METHOD PROTECTED OnExecErrorClear : DINT
VAR_IN_OUT
  /// Robot assignment of function
  AxesGroup : AxesGroup; 
END_VAR
                  OnExecErrorClear := Reset();
                
END_METHOD

METHOD PROTECTED OnExecRun : DINT
VAR_IN_OUT
  /// Robot assignment of function
  AxesGroup : AxesGroup; 
END_VAR
                  
                
END_METHOD

METHOD PROTECTED OnExecStart : DINT
VAR_IN_OUT
  /// Robot assignment of function
  AxesGroup : AxesGroup; 
END_VAR
                  
                
END_METHOD

METHOD PROTECTED OnUpdateStateFlags
VAR_INPUT
  /// Command message state
  State : CmdMessageState;
END_VAR
                  // Reset State flags
Done := FALSE;

CASE State OF

  // No operation or process is active
  CmdMessageState.EMPTY               :;
  // Created but not yet started
  CmdMessageState.CREATED             :;
  // Buffered and awaiting execution
  CmdMessageState.BUFFERED            :;
  // Buffered in planner for future execution
  CmdMessageState.BUFFERED_IN_PLANNER :;
  // Currently active and in progress
  CmdMessageState.ACTIVE              :;
  // Interrupted and awaiting continuation
  CmdMessageState.INTERRUPTED         :;
  // Requested for abort
  CmdMessageState.ABORT_REQUEST       :;
  // Successfully completed
  CmdMessageState.DONE                : Done := TRUE;
                                        Busy := FALSE;
  // Aborted before completion
  CmdMessageState.ABORTED             : Busy := FALSE;
  // Encountered an error during execution
  CmdMessageState.ERROR               : Error := TRUE;
                                        Busy  := FALSE;
END_CASE
                
END_METHOD

METHOD PROTECTED Reset : DINT
VAR_INPUT
END_VAR
                  Reset := SUPER^.Reset();

Done := FALSE;
Busy := FALSE;
                
END_METHOD
END_FUNCTION_BLOCK

FUNCTION_BLOCK RobotLibraryBaseFB EXTENDS RobotLibraryLogFB
// ------------------------------------------------------------------------- 
//  SRCI Robot Library                                                
// ------------------------------------------------------------------------- 
//                                                                           
//  Object:      RobotLibraryBaseFB                                       
//  Author:      Thorsten Brach                                                
//  Date:        2024-06-01
//
//  Description:                                              
//   
//                                                                           
//  Copyright: 
//    (C) 2024 Thorsten Brach. All rights reserved                                                                                                                                            
//             Licensed under the MIT License.
//                                                                           
//  Disclaimer:                                                                           
//    This project is provided without any guarantee and can be used for   
//    private and commercial purposes. Any use is at the user’s 
//    own risk and responsibility.
//
// -------------------------------------------------------------------------
VAR_INPUT
  /// User defined command name
  Name         : STRING(80);
  /// Execution Mode
  ExecMode     : ExecutionMode;
  /// Priority
  Priority     : PriorityLevel;
END_VAR
VAR_OUTPUT
  /// Command data
  CommandData  : RobotLibraryCommandDataFB;
  /// response data
  ResponseData : RobotLibraryResponseDataFB;
  /// An error occurred during the execution of the command
  Error        : BOOL;
  /// ErrorID reported by RC for error identification according to Table 7-1
  ErrorID      : WORD;
  ErrorIdEnum  : RobotLibraryErrorIdEnum;  
  ErrorAddTxt  : STRING(RobotLibraryConstants.MAX_ADD_TEXT_LENGTH);
  
  /// WarningID for warning identification reported during execution of command according to Table 7-3
  WarningID    : WORD;
  WarningIdEnum: RobotLibraryWarningIdEnum;  
  /// InfoID for info identification reported during execution of command according to Table 7-5
  InfoID       : WORD;    
  InfoIdEnum   : RobotLibraryInfoIdEnum;  
END_VAR
VAR_IN_OUT
  /// Robot assignment of function
  AxesGroup    : AxesGroup; 
END_VAR

VAR
  /// Rising edge for error
  {attribute 'hide'}
 _error_R                  : R_TRIG;
  /// Rising edge for warning
  {attribute 'hide'}
 _warning_R                : R_TRIG;
  /// Rising edge for information
  {attribute 'hide'}
 _info_R                   : R_TRIG;
  /// clear error active
 _clearError               : BOOL;
  /// cancel active
 _cancel                   : BOOL; 
  /// unique ID
 _uniqueID                 : UDINT;  
  /// flag for response received
 _responseReceived         : BOOL;
  /// internal step counter
 _stepCmd                  : DINT;
  /// internal timer  
  {attribute 'hide'}
 _timerCmd                 : TON;
  /// internal timeout 
  {attribute 'hide'}
 _timeoutCmd               : TIME := T#5S;
  /// internal step counter for ClearError
 _stepClearError           : DINT;
  /// internal timer for ClearError
  {attribute 'hide'}
 _timerClearError          : TON;
  /// internal timeout for ClearError 
  {attribute 'hide'}
 _timeoutClearError        : TIME := T#5S;

  /// internal step counter for Cancel
 _stepCancel               : DINT;
  /// internal timer for Cancel  
  {attribute 'hide'}
 _timerCancel              : TON;
  /// internal timeout for Cancel 
  {attribute 'hide'}
 _timeoutCancel            : TIME := T#5S;

  /// internal command header
 _cmdHeader                : CmdHeader;  
  /// internal response header
 _rspHeader                : RspHeader;
  /// internal flag for send a parameter update
 _parameterUpdateInternal  : BOOL; 
  /// internal flag for parameter has changed
 _parameterChanged         : BOOL;
  /// internal flag for parameter are valid
 _parameterValid           : BOOL;
END_VAR

            OnCall               (AxesGroup := AxesGroup);
OnExecRun            (AxesGroup := AxesGroup);
CheckParameterChanged(AxesGroup := AxesGroup);


IF ( AxesGroup.State.OnlineChange_R.Q )
THEN
  OnOnlineChange(AxesGroup := AxesGroup);
END_IF
          

METHOD PUBLIC CallBack : DINT
VAR_INPUT
  /// Response data
  RspData   : AxesGroupAcyclicAcrEntryRspBuffer;  
  /// Timestamp
  Timestamp : SystemTime;
END_VAR
                  // Create log entry
CreateLogMessagePara2 ( Timestamp   := Timestamp,
                        MessageType := MessageType.CMD,
                        Severity    := Severity.DEBUG,
                        MessageCode := 0,
                        MessageText := 'Callback reveiced in FB {1} <{2}>',
                        Para1       := MyType,
                        Para2       := Name);

                   
                   
ResponseData.Reset();
ResponseData.Payload    := RspData.Payload; 
ResponseData.PayloadLen := RspData.PayloadLen;
ParseResponsePayload( ResponseData :=  ResponseData , Timestamp := Timestamp);

// set flag for response received
_responseReceived := TRUE;
                
END_METHOD

METHOD PROTECTED CheckFunctionSupported : BOOL
VAR_IN_OUT
  /// Robot assignment of function
  AxesGroup : AxesGroup; 
END_VAR
                  Error       := TRUE;
ErrorID     := RobotLibraryErrorIdEnum.ERR_FUNCTION_NOT_SUPPORTED;
ErrorAddTxt := CONCAT(THIS^._myType, ' ');
ErrorAddTxt := CONCAT(ErrorAddTxt , THIS^.Name);


// Create log entry
CreateLogMessagePara1 ( Timestamp   := AxesGroup.State.SystemTime,
                        MessageType := MessageType.CMD,
                        Severity    := Severity.DEBUG,
                        MessageCode := 0,
                        MessageText := 'Execution canceled, because function <{1}> is not supported by the robot controller',
                        Para1       :=  _myType);
                
END_METHOD

METHOD PROTECTED CheckParameterChanged : BOOL
VAR_IN_OUT
  /// Robot assignment of function
  AxesGroup    : AxesGroup; 
END_VAR
                  IF ( CheckParameterChanged )
THEN
  AxesGroup.Acyclic.ActiveCommandRegister.NotifyParameterChanged := _uniqueID;
END_IF
                
END_METHOD

METHOD PROTECTED CheckParameterValid : BOOL
VAR_IN_OUT
  /// Robot assignment of function
  AxesGroup : AxesGroup; 
END_VAR
                  CheckParameterValid := TRUE;
                
END_METHOD

METHOD INTERNAL CreateCommandPayload : RobotLibraryCommandDataFB
VAR_IN_OUT
  /// Robot assignment of function
  AxesGroup    : AxesGroup; 
END_VAR
                  // Reset all variables
CreateCommandPayload.Reset();
// Add CmdType
CreateCommandPayload.AddUint(_cmdHeader.CmdTyp);
// Add Reserve_ExecMode
CreateCommandPayload.AddHalfBytes(  0               , _cmdHeader.ExecMode);
// Add ParSeq_Priority
CreateCommandPayload.AddHalfBytes( _cmdHeader.ParSeq, _cmdHeader.Priority);
                
END_METHOD

METHOD PROTECTED OnApplyOutCmd
VAR_INPUT
  /// Command message state
  State : CmdMessageState;
END_VAR
                  
                
END_METHOD

METHOD PROTECTED OnCall
VAR_IN_OUT
  /// Robot assignment of function
  AxesGroup : AxesGroup; 
END_VAR
                  // map numeric value to enum, so that the corresponding message text is directly shown by the tooltip
ErrorIdEnum   := ErrorId;
WarningIdEnum := WarningId;
InfoIdEnum    := InfoId;

Error := ErrorID <> RobotLibraryConstants.OK;

InternalLogger   := AxesGroup.MessageLog; 
ExternalLogger   := AxesGroup.MessageLog.ExternalLogger;
LogLevel         := AxesGroup.MessageLog.LogLevel;

// building rising edges for error, warning, info number detected
_error_R  ( CLK := ErrorID   <> RobotLibraryConstants.OK );
_warning_R( CLK := WarningID <> RobotLibraryConstants.OK );
_info_R   ( CLK := InfoID    <> RobotLibraryConstants.OK );


// Log Command events to message log 
IF  ( LogLevel < _rspHeader.AlarmMessageSeverity ) AND
   (( _error_R  .Q                               ) OR 
    ( _warning_R.Q                               ) OR 
    ( _info_R   .Q                               ))
THEN
  // Add command message to message buffer       
  AxesGroup.MessageLog
    .AddMessageLogByParameter(  Timestamp   :=   AxesGroup.State.SystemTime,
                                MessageType :=   MessageType.CMD,
                                MessageCode :=  _rspHeader.AlarmMessageCode,
                                MessageText :=   CONCAT(MyType, CONCAT(' : ' , MESSAGE_CODE_TO_STRING(_rspHeader.AlarmMessageCode))),
                                Severity    :=  _rspHeader.AlarmMessageSeverity ); 
END_IF 


IF ( _error_R.Q)
THEN
  // Create log entry
  CreateLogMessagePara2 ( Timestamp   := AxesGroup.State.SystemTime,
                          MessageType := MessageType.CMD,
                          Severity    := Severity.DEBUG,
                          MessageCode := 0,
                          MessageText := 'Error with ID: 16#{1} in FB {2} received ',
                          Para1       := WORD_TO_STRING_HEX(ErrorID),
                          Para2       := MyType);                        
END_IF

IF ( _warning_R.Q)
THEN
  // Create log entry
  CreateLogMessagePara2 ( Timestamp   := AxesGroup.State.SystemTime,
                          MessageType := MessageType.CMD,
                          Severity    := Severity.DEBUG,
                          MessageCode := 0,
                          MessageText := 'Warning with ID: 16#{1} in FB {2} received ',
                          Para1       := WORD_TO_STRING_HEX(WarningID),
                          Para2       := MyType);                        
END_IF

IF ( _info_R.Q)
THEN
  // Create log entry
  CreateLogMessagePara2 ( Timestamp   := AxesGroup.State.SystemTime,
                          MessageType := MessageType.CMD,
                          Severity    := Severity.DEBUG,
                          MessageCode := 0,
                          MessageText := 'Info with ID: 16#{1} in FB {2} received ',
                          Para1       := WORD_TO_STRING_HEX(InfoID),
                          Para2       := MyType);                        
END_IF
                
END_METHOD

METHOD PROTECTED OnExecRun : DINT
VAR_IN_OUT
  /// Robot assignment of function
  AxesGroup : AxesGroup; 
END_VAR
                  
                
END_METHOD

METHOD OnOnlineChange : DINT
VAR_IN_OUT
  /// Robot assignment of function
  AxesGroup : AxesGroup; 
END_VAR
                  // update pointer to command FB
AxesGroup.Acyclic.ActiveCommandRegister.OnOnlineChange( UniqueID := _uniqueID, pCommandFB := ADR(THIS^));
                
END_METHOD

METHOD PROTECTED OnUpdateStateFlags
VAR_INPUT
  /// Command message state
  State : CmdMessageState;
END_VAR
                  
                
END_METHOD

METHOD INTERNAL ParseResponsePayload : DINT
VAR_INPUT
  /// Response data
  ResponseData : RobotLibraryResponseDataFB;
  /// Timestamp
  Timestamp    : SystemTime;  
END_VAR
                  // reset message IDs 
InfoID    := 0;
WarningID := 0;
ErrorID   := 0;

// get State
_rspHeader.State                := ResponseData.GetHalfeByte1(IncPayloadPtr := FALSE);
// get ParSeq
_rspHeader.ParSeq               := ResponseData.GetHalfeByte2(IncPayloadPtr := TRUE);
// get AlarmMessageSeverity
_rspHeader.AlarmMessageSeverity := ResponseData.GetSint();
// get AlarmMessageCode
_rspHeader.AlarmMessageCode     := ResponseData.GetUint();


// Update InfoID / WarningID / ErrorID
CASE _rspHeader.AlarmMessageSeverity OF

  // Informative message
  Severity.INFO        : SetInfo   ( InfoID    := _rspHeader.AlarmMessageCode, Overwrite := TRUE );
  // Warning message
  Severity.WARNING     : SetWarning( WarningID := _rspHeader.AlarmMessageCode, Overwrite := TRUE );
  // Error message
  Severity.ERROR       : SetError  ( ErrorID   := _rspHeader.AlarmMessageCode, Overwrite := TRUE ); 
  // Fataö error message
  Severity.FATAL_ERROR : SetError  ( ErrorID   := _rspHeader.AlarmMessageCode, Overwrite := TRUE );

END_CASE

ParseResponsePayload := ResponseData.PayloadPtr;
                
END_METHOD

METHOD PROTECTED Reset : DINT
VAR_INPUT
END_VAR
                  _parameterUpdateInternal := FALSE;
_responseReceived := FALSE;

_uniqueId := 0;
_stepCmd  := 0;
Error     := FALSE;
ErrorID   := 0;
WarningID := 0;
InfoID    := 0;  

Reset := RobotLibraryConstants.OK;
                
END_METHOD

METHOD PUBLIC SetError
VAR_INPUT
  /// ErrorID reported by RC for error identification according to Table 7-1
  ErrorID   : WORD;
  /// TRUE = overwrite an existing error 
  Overwrite : BOOL;
END_VAR
                  IF ( NOT HasError ) OR ( Overwrite )
THEN
  THIS^.ErrorID := ErrorID;
END_IF
                
END_METHOD

METHOD PUBLIC SetInfo
VAR_INPUT
  /// InfoID for info identification reported during execution of command according to Table 7-5
  InfoID    : WORD;
  /// TRUE = overwrite an existing info 
  Overwrite : BOOL;
END_VAR
                  IF ( NOT HasInfo ) OR ( Overwrite )
THEN
  THIS^.InfoID := InfoID;
END_IF
                
END_METHOD

METHOD PUBLIC SetWarning
VAR_INPUT
  /// WarningID for warning identification reported during execution of command according to Table 7-3
  WarningID : WORD;
  /// TRUE = overwrite an existing warning 
  Overwrite : BOOL;
END_VAR
                  IF ( NOT HasWarning ) OR ( Overwrite )
THEN
  THIS^.WarningID := WarningID;
END_IF
                
END_METHOD

PROPERTY PUBLIC HasError : Bool
GET
VAR
END_VAR
                    HasError := ErrorID <> RobotLibraryErrorIdEnum.NO_ERROR;
                  
END_GET
END_PROPERTY

PROPERTY PUBLIC HasInfo : BOOL
GET
VAR
END_VAR
                    HasInfo := InfoID <> RobotLibraryInfoIdEnum.NO_INFO;
                  
END_GET
END_PROPERTY

PROPERTY PUBLIC HasWarning : BOOL
GET
VAR
END_VAR
                    HasWarning := WarningID <> RobotLibraryWarningIdEnum.NO_WARNING;
                  
END_GET
END_PROPERTY
END_FUNCTION_BLOCK

FUNCTION_BLOCK RobotLibraryLogFB
// ------------------------------------------------------------------------- 
//  SRCI Robot Library                                                
// ------------------------------------------------------------------------- 
//                                                                           
//  Object:      RobotLibraryLogFB                                       
//  Author:      Thorsten Brach                                                
//  Date:        2024-11-10
//
//  Description:                                              
//   
//                                                                           
//  Copyright: 
//    (C) 2024 Thorsten Brach. All rights reserved                                                                                                                                            
//             Licensed under the MIT License.
//                                                                           
//  Disclaimer:                                                                           
//    This project is provided without any guarantee and can be used for   
//    private and commercial purposes. Any use is at the user’s 
//    own risk and responsibility.
//
// -------------------------------------------------------------------------
VAR_INPUT
  /// Interface to an internal logger
  InternalLogger : IMessageLogger;  
  /// Interface to an external logger
  ExternalLogger : IMessageLogger;  
  /// Logging level
  LogLevel       : LogLevelEnum := LogLevelEnum.INFO; 
END_VAR

VAR
  /// Type of the function block
 _myType         : STRING;
END_VAR

            
          

METHOD CreateLogMessage : STRING(RobotLibraryParameter.MESSAGE_TEXT_LEN)
VAR_INPUT
  /// Timestamp
  Timestamp   : SystemTime;
  /// Type of message according to Table 5-46:
  MessageType : MessageType;
  /// Severity of message according to Table 5-47: Debug, Info, Warning, Error, Fatal error
  Severity    : Severity;
  /// Code of messages
  MessageCode : DWORD;
  /// Static text of message
  MessageText : STRING(RobotLibraryParameter.MESSAGE_TEXT_LEN);  
END_VAR

VAR
  /// internal log message 
 _message    : AlarmMessage;
  /// internal string
 _tmpString  : STRING(255);
END_VAR
                  IF ( LogLevel <= Severity )
THEN
 _message.Timestamp   := Timestamp;
 _message.MessageType := MessageType;
 _message.Severity    := Severity;
 _message.MessageCode := MessageCode;
 _message.MessageText := StrPadRight(MyType,' ', RobotLibraryDefines.MaxTypeNameLength);
 _message.MessageText := CONCAT(_message.MessageText, ': ');
 _message.MessageText := CONCAT(_message.MessageText,MessageText);

  // return log message
  CreateLogMessage := ALARM_MESSAGE_TO_STRING(_message);
  
  // Check internal logger valid ? 
  IF ( InternalLogger <> 0 )
  THEN  
    InternalLogger.AddSystemLog( SystemLog := ALARM_MESSAGE_TO_STRING(_message));
  END_IF

  // Check external logger valid ? 
  IF ( ExternalLogger <> 0 )
  THEN  
    ExternalLogger.AddSystemLog( SystemLog := ALARM_MESSAGE_TO_STRING(_message));
  END_IF
END_IF
                
END_METHOD

METHOD CreateLogMessagePara1 : STRING(RobotLibraryParameter.MESSAGE_TEXT_LEN)
VAR_INPUT
  /// Timestamp
  Timestamp   : SystemTime;
  /// Type of message according to Table 5-46:
  MessageType : MessageType;
  /// Severity of message according to Table 5-47: Debug, Info, Warning, Error, Fatal error
  Severity    : Severity;
  /// Code of messages
  MessageCode : DWORD;
  /// Static text of message
  MessageText : STRING(RobotLibraryParameter.MESSAGE_TEXT_LEN);  
  /// sub string which will replace the placeholder {1}
  Para1       : STRING(RobotLibraryParameter.MESSAGE_TEXT_LEN);
END_VAR
VAR
  /// internal log message 
 _logMessage : AlarmMessage;
END_VAR
                  IF ( LogLevel <= Severity )
THEN
  MessageText := StrReplace(MessageText,'{1}', Para1);
  
  CreateLogMessagePara1 
    := CreateLogMessage( Timestamp   := Timestamp,
                         MessageType := MessageType,
                         Severity    := Severity,
                         MessageCode := MessageCode,
                         MessageText := MessageText);
END_IF                         
                
END_METHOD

METHOD CreateLogMessagePara2 : STRING(RobotLibraryParameter.MESSAGE_TEXT_LEN)
VAR_INPUT
  /// Timestamp
  Timestamp   : SystemTime;
  /// Type of message according to Table 5-46:
  MessageType : MessageType;
  /// Severity of message according to Table 5-47: Debug, Info, Warning, Error, Fatal error
  Severity    : Severity;
  /// Code of messages
  MessageCode : DWORD;
  /// Static text of message
  MessageText : STRING(RobotLibraryParameter.MESSAGE_TEXT_LEN);  
  /// sub string which will replace the placeholder {1}
  Para1       : STRING(RobotLibraryParameter.MESSAGE_TEXT_LEN);
  /// sub string which will replace the placeholder {2}
  Para2       : STRING(RobotLibraryParameter.MESSAGE_TEXT_LEN);
END_VAR
VAR
  /// internal log message 
 _logMessage : AlarmMessage;
END_VAR
                  IF ( LogLevel <= Severity )
THEN
  MessageText := StrReplace(MessageText,'{2}', Para2);
  
  CreateLogMessagePara2 
    := CreateLogMessagePara1( Timestamp   := Timestamp,
                              MessageType := MessageType,
                              Severity    := Severity,
                              MessageCode := MessageCode,
                              MessageText := MessageText,
                              Para1       := Para1);
END_IF                              
                
END_METHOD

METHOD CreateLogMessagePara3 : STRING(RobotLibraryParameter.MESSAGE_TEXT_LEN)
VAR_INPUT
  /// Timestamp
  Timestamp   : SystemTime;
  /// Type of message according to Table 5-46:
  MessageType : MessageType;
  /// Severity of message according to Table 5-47: Debug, Info, Warning, Error, Fatal error
  Severity    : Severity;
  /// Code of messages
  MessageCode : DWORD;
  /// Static text of message
  MessageText : STRING(RobotLibraryParameter.MESSAGE_TEXT_LEN);  
  /// sub string which will replace the placeholder {1}
  Para1       : STRING(RobotLibraryParameter.MESSAGE_TEXT_LEN);
  /// sub string which will replace the placeholder {2}
  Para2       : STRING(RobotLibraryParameter.MESSAGE_TEXT_LEN);
  /// sub string which will replace the placeholder {3}
  Para3       : STRING(RobotLibraryParameter.MESSAGE_TEXT_LEN);
END_VAR
VAR
  /// internal log message 
 _logMessage : AlarmMessage;
END_VAR
                  IF ( LogLevel <= Severity )
THEN
  MessageText := StrReplace(MessageText,'{3}', Para3);
  
  CreateLogMessagePara3
    := CreateLogMessagePara2( Timestamp   := Timestamp,
                              MessageType := MessageType,
                              Severity    := Severity,
                              MessageCode := MessageCode,
                              MessageText := MessageText,
                              Para1       := Para1,
                              Para2       := Para2);
END_IF                              
                
END_METHOD

METHOD CreateLogMessagePara4 : STRING(RobotLibraryParameter.MESSAGE_TEXT_LEN)
VAR_INPUT
  /// Timestamp
  Timestamp   : SystemTime;
  /// Type of message according to Table 5-46:
  MessageType : MessageType;
  /// Severity of message according to Table 5-47: Debug, Info, Warning, Error, Fatal error
  Severity    : Severity;
  /// Code of messages
  MessageCode : DWORD;
  /// Static text of message
  MessageText : STRING(RobotLibraryParameter.MESSAGE_TEXT_LEN);  
  /// sub string which will replace the placeholder {1}
  Para1       : STRING(RobotLibraryParameter.MESSAGE_TEXT_LEN);
  /// sub string which will replace the placeholder {2}
  Para2       : STRING(RobotLibraryParameter.MESSAGE_TEXT_LEN);
  /// sub string which will replace the placeholder {3}
  Para3       : STRING(RobotLibraryParameter.MESSAGE_TEXT_LEN);
  /// sub string which will replace the placeholder {4}
  Para4       : STRING(RobotLibraryParameter.MESSAGE_TEXT_LEN);
END_VAR
VAR
  /// internal log message 
 _logMessage : AlarmMessage;
END_VAR
                  IF ( LogLevel <= Severity )
THEN
  MessageText := StrReplace(MessageText,'{4}', Para4);
  
  CreateLogMessagePara4
    := CreateLogMessagePara3( Timestamp   := Timestamp,
                              MessageType := MessageType,
                              Severity    := Severity,
                              MessageCode := MessageCode,
                              MessageText := MessageText,
                              Para1       := Para1,
                              Para2       := Para2,
                              Para3       := Para3);
END_IF                              
                
END_METHOD

METHOD CreateLogMessagePara5 : STRING(RobotLibraryParameter.MESSAGE_TEXT_LEN)
VAR_INPUT
  /// Timestamp
  Timestamp   : SystemTime;
  /// Type of message according to Table 5-46:
  MessageType : MessageType;
  /// Severity of message according to Table 5-47: Debug, Info, Warning, Error, Fatal error
  Severity    : Severity;
  /// Code of messages
  MessageCode : DWORD;
  /// Static text of message
  MessageText : STRING(RobotLibraryParameter.MESSAGE_TEXT_LEN);  
  /// sub string which will replace the placeholder {1}
  Para1       : STRING(RobotLibraryParameter.MESSAGE_TEXT_LEN);
  /// sub string which will replace the placeholder {2}
  Para2       : STRING(RobotLibraryParameter.MESSAGE_TEXT_LEN);
  /// sub string which will replace the placeholder {3}
  Para3       : STRING(RobotLibraryParameter.MESSAGE_TEXT_LEN);
  /// sub string which will replace the placeholder {4}
  Para4       : STRING(RobotLibraryParameter.MESSAGE_TEXT_LEN);
  /// sub string which will replace the placeholder {5}
  Para5       : STRING(RobotLibraryParameter.MESSAGE_TEXT_LEN);
END_VAR
VAR
  /// internal log message 
 _logMessage : AlarmMessage;
END_VAR
                  IF ( LogLevel <= Severity )
THEN  
  MessageText := StrReplace(MessageText,'{5}', Para5);
  
  CreateLogMessagePara5
    := CreateLogMessagePara4( Timestamp   := Timestamp,
                              MessageType := MessageType,
                              Severity    := Severity,
                              MessageCode := MessageCode,
                              MessageText := MessageText,
                              Para1       := Para1,
                              Para2       := Para2,
                              Para3       := Para3,
                              Para4       := Para4);
END_IF                              
                
END_METHOD

METHOD CreateLogMessagePara6 : STRING(RobotLibraryParameter.MESSAGE_TEXT_LEN)
VAR_INPUT
  /// Timestamp
  Timestamp   : SystemTime;
  /// Type of message according to Table 5-46:
  MessageType : MessageType;
  /// Severity of message according to Table 5-47: Debug, Info, Warning, Error, Fatal error
  Severity    : Severity;
  /// Code of messages
  MessageCode : DWORD;
  /// Static text of message
  MessageText : STRING(RobotLibraryParameter.MESSAGE_TEXT_LEN);  
  /// sub string which will replace the placeholder {1}
  Para1       : STRING(RobotLibraryParameter.MESSAGE_TEXT_LEN);
  /// sub string which will replace the placeholder {2}
  Para2       : STRING(RobotLibraryParameter.MESSAGE_TEXT_LEN);
  /// sub string which will replace the placeholder {3}
  Para3       : STRING(RobotLibraryParameter.MESSAGE_TEXT_LEN);
  /// sub string which will replace the placeholder {4}
  Para4       : STRING(RobotLibraryParameter.MESSAGE_TEXT_LEN);
  /// sub string which will replace the placeholder {5}
  Para5       : STRING(RobotLibraryParameter.MESSAGE_TEXT_LEN);
  /// sub string which will replace the placeholder {6}
  Para6       : STRING(RobotLibraryParameter.MESSAGE_TEXT_LEN);
END_VAR
VAR
  /// internal log message 
 _logMessage : AlarmMessage;
END_VAR
                  IF ( LogLevel <= Severity )
THEN
  MessageText := StrReplace(MessageText,'{6}', Para6);
  
  CreateLogMessagePara6
    := CreateLogMessagePara5( Timestamp   := Timestamp,
                              MessageType := MessageType,
                              Severity    := Severity,
                              MessageCode := MessageCode,
                              MessageText := MessageText,
                              Para1       := Para1,
                              Para2       := Para2,
                              Para3       := Para3,
                              Para4       := Para4,
                              Para5       := Para5);
END_IF                       
                
END_METHOD

PROPERTY PROTECTED MyType : STRING
GET
VAR
END_VAR
                    MyType := _myType;
                  
END_GET
SET
VAR
END_VAR
                    _myType := MyType;

// set the max type name length 
RobotLibraryDefines.MaxTypeNameLength := MAX(LEN(_myType), RobotLibraryDefines.MaxTypeNameLength);
                  
END_SET
END_PROPERTY
END_FUNCTION_BLOCK

FUNCTION_BLOCK AxesGroupMessageLogFB IMPLEMENTS IMessageLogger
// ------------------------------------------------------------------------- 
//  SRCI Robot Library                                                
// ------------------------------------------------------------------------- 
//                                                                           
//  Object:      AxesGroupMessageLogFB                                       
//  Author:      Thorsten Brach                                                
//  Date:        2025-01-05
//
//  Description:                                              
//   
//                                                                           
//  Copyright: 
//    (C) 2025 Thorsten Brach. All rights reserved                                                                                                                                            
//             Licensed under the MIT License.
//                                                                           
//  Disclaimer:                                                                           
//    This project is provided without any guarantee and can be used for   
//    private and commercial purposes. Any use is at the user’s 
//    own risk and responsibility.
//
// -------------------------------------------------------------------------
VAR_INPUT
  /// Logging level
  LogLevel         : LogLevel;
  /// Interface to an external logger
  ExternalLogger   : IMessageLogger;
END_VAR


VAR_OUTPUT
  /// Amount of system log entries
  SystemLogEntries : UINT := 0;
  /// Amount of message log entries
  MessagesEntries  : UINT := 0;
  /// System log
  SystemLogs       : ARRAY[0..RobotLibraryParameter.SYSTEM_LOG_MAX ] OF STRING(RobotLibraryParameter.MESSAGE_TEXT_LEN);
  /// Message Log
  Messages         : ARRAY[0..RobotLibraryParameter.MESSAGE_LOG_MAX] OF AlarmMessage;  
END_VAR

            
          

METHOD PUBLIC AddMessageLog
VAR_INPUT
  MessageLog : AlarmMessage;
END_VAR

VAR
  /// internal index
 _idx            : DINT;
  /// internal index to delete
 _idxFound       : DINT;
  /// lowest Severity
 _lowestSeverity : Severity := Severity.FATAL_ERROR;
  /// temporary buffer ( must be one element less than the message log !!! )
 _tmpBuffer      : ARRAY[0..RobotLibraryParameter.MESSAGE_LOG_MAX -1] OF AlarmMessage; 
END_VAR
                  // Check entry must be added ? 
IF (( LogLevel  <= MessageLog.Severity     ) AND
    ( LogLevel  >  LogLevelEnum.DEACTIVATE ))
THEN
  // Check message buffer is full ? 
  IF ( MessagesEntries >= RobotLibraryParameter.MESSAGE_LOG_MAX )
  THEN
    // find lowest Severity
    FOR _idx := 1 TO RobotLibraryParameter.MESSAGE_LOG_MAX
    DO
      // check entry has a lower severity ? 
     _lowestSeverity := MIN( Messages[_idx].Severity, _lowestSeverity );
		END_FOR

    // search for the oldes message with a lower Severity 
    FOR _idx := RobotLibraryParameter.MESSAGE_LOG_MAX TO 1 BY -1
    DO
      // message found ?
      IF (( Messages[_idx].Severity <   MessageLog.Severity ) AND
          ( Messages[_idx].Severity <= _lowestSeverity      ))
      THEN
        // save index to delete 
       _idxFound := _idx;
        EXIT;
			END_IF
		END_FOR
    
    // check message must be deleted ? 
    IF ( _idxFound > 0 )
    THEN
      // shift all messages starting from the found index one position forwards
      FOR _idx := _idxFound TO RobotLibraryParameter.MESSAGE_LOG_MAX -1
      DO
        Messages[_idx] := Messages[_idx +1];
			END_FOR
		END_IF
  END_IF  

  // shift all messages one position backwards
  // shift messages log entries
  SysDepMemCpy( pDest := ADR(_tmpBuffer[0]), pSrc := ADR(  Messages[0]), DataLen := SIZEOF(_tmpBuffer));
  SysDepMemCpy( pDest := ADR(  Messages[1]), pSrc := ADR(_tmpBuffer[0]), DataLen := SIZEOF(_tmpBuffer));
  
  
  // Add new message 
  Messages[0].Timestamp   := MessageLog.Timestamp;           
  Messages[0].MessageType := MessageLog.MessageType;
  Messages[0].Severity    := MessageLog.Severity;
  Messages[0].MessageText := MessageLog.MessageText;
  Messages[0].MessageCode := MessageLog.MessageCode;
  
  // inc message counter
  MessagesEntries := DINT_TO_UINT(LIMIT(0, MessagesEntries + 1, RobotLibraryParameter.MESSAGE_LOG_MAX));
END_IF
                
END_METHOD

METHOD Public AddMessageLogByParameter
VAR_INPUT
  /// Timestamp
  Timestamp   : SystemTime;
  /// Type of message according to Table 5-46:
  MessageType : MessageType;
  /// Severity of message according to Table 5-47: Debug, Info, Warning, Error, Fatal error
  Severity    : Severity;
  /// Code of messages
  MessageCode : DWORD;
  /// Static text of message
  MessageText : STRING(RobotLibraryParameter.MESSAGE_TEXT_LEN);    
END_VAR

VAR
  /// temporary message 
 _message : AlarmMessage;
END_VAR
                  _message.Timestamp   := Timestamp;
_message.MessageType := MessageType;
_message.MessageCode := MessageCode;
_message.MessageText := MessageText;
_message.Severity    := Severity;

// Add message to message buffer       
AddMessageLog(_message);        
                
END_METHOD

METHOD PUBLIC AddSystemLog
VAR_INPUT
  /// system log message
  SystemLog : STRING(255);
END_VAR
VAR
  /// internal index
 _idx       : DINT;
  /// internal log message 
 _message   : AlarmMessage;
  /// temporary buffer ( must be one element less than the system log !!! )
 _tmpBuffer : ARRAY[0..RobotLibraryParameter.SYSTEM_LOG_MAX -1] OF STRING(RobotLibraryParameter.MESSAGE_TEXT_LEN);
END_VAR
                  // shift system log entries
SysDepMemCpy( pDest := ADR(_tmpBuffer[0]), pSrc := ADR(SystemLogs[0]), DataLen := SIZEOF(_tmpBuffer));
SysDepMemCpy( pDest := ADR(SystemLogs[1]), pSrc := ADR(_tmpBuffer[0]), DataLen := SIZEOF(_tmpBuffer));

// Delete CR from system log message
SystemLog := StrReplace(SystemLog, '$R', '');
// Delete LF from system log message          
SystemLog := StrReplace(SystemLog, '$N', '');    
       
// Add System log to buffer 
SystemLogs[0] := SystemLog;
 
// inc SystemLog counter
SystemLogEntries := DINT_TO_UINT(LIMIT(0, SystemLogEntries + 1, RobotLibraryParameter.SYSTEM_LOG_MAX));
                
END_METHOD

METHOD CheckMessageCodePresent : BOOL
VAR_INPUT
  /// Code of messages
  MessageCode : DWORD;
END_VAR

VAR
  /// internal index for loops
 _idx : DINT;
END_VAR
                  FOR _idx := 0 TO RobotLibraryParameter.MESSAGE_LOG_MAX
DO
  IF (Messages[_idx].MessageCode = MessageCode)
  THEN
    CheckMessageCodePresent := TRUE;
    RETURN;
	END_IF
END_FOR
                
END_METHOD

METHOD PUBLIC DeleteMessages
VAR_INPUT
END_VAR
                  // reset messages
SysDepMemSet(ADR(Messages), 0, SIZEOF(Messages));
// reset message counter
MessagesEntries := 0;
                
END_METHOD

METHOD DeleteSystemLogs
VAR_INPUT
END_VAR
                  // reset SystemLogs
SysDepMemSet(ADR(SystemLogs), 0, SIZEOF(SystemLogs));
// reset SystemLogs counter
SystemLogEntries := 0;
                
END_METHOD
END_FUNCTION_BLOCK

{attribute 'pack_mode' := '1'} 
FUNCTION_BLOCK RobotLibraryRecvDataBaseFB
// ------------------------------------------------------------------------- 
//  SRCI Robot Library                                                
// ------------------------------------------------------------------------- 
//                                                                           
//  Object:      RobotLibraryRecvDataFB                                       
//  Author:      Thorsten Brach                                                
//  Date:        2024-06-01
//
//  Description:                                              
//   
//                                                                           
//  Copyright: 
//    (C) 2024 Thorsten Brach. All rights reserved                                                                                                                                            
//             Licensed under the MIT License.
//                                                                           
//  Disclaimer:                                                                           
//    This project is provided without any guarantee and can be used for   
//    private and commercial purposes. Any use is at the user’s 
//    own risk and responsibility.
//
// -------------------------------------------------------------------------
VAR_INPUT
  /// Payload length
  PayloadLen : UDINT;
  /// Payload pointer
  PayloadPtr : DINT;
END_VAR

VAR
  /// internal pointer to payload 
  pPayload : POINTER TO BYTE;
END_VAR

            
          

/// returns a ArmConfigParameter from the payload buffer from the current payload pointer address and increase the payload pointer afterwards
METHOD GetArmConfig : ArmConfigParameter
VAR
  /// temporary byte
 _tmpByte : BYTE;
END_VAR
// Table 5-17: Meaning of “Config” byte
// BIT 0 Shoulder TRUE : Shoulder is Back
//                FALSE: Shoulder is Front
// BIT 1 Elbow    TRUE : Elbow is Down
//                FALSE: Elbow is Up
// BIT 2 Wrist    TRUE : Wrist is Flip
//                FALSE: Wrist is Non-Flip
// BIT 3 Spare Not used
// BIT 4 Spare Not Used
// BIT 5 Spare Not Used
// BIT 6 Spare Not Used
// BIT 7 Spare Not Used
                  // get 1st Byte
_tmpByte := GetByte();

IF ( _tmpByte.0 ) 
THEN
  GetArmConfig.Shoulder := ArmConfigShoulder.BACK;
ELSE
  GetArmConfig.Shoulder := ArmConfigShoulder.FRONT;
END_IF

IF ( _tmpByte.1 ) 
THEN
  GetArmConfig.Elbow := ArmConfigElbow.DOWN;
ELSE
  GetArmConfig.Elbow := ArmConfigElbow.UP;
END_IF

IF ( _tmpByte.2 ) 
THEN
  GetArmConfig.Wrist := ArmConfigWrist.FLIP;
ELSE
  GetArmConfig.Wrist := ArmConfigWrist.NON_FLIP;
END_IF


// get 2nd byte to inc the PayloadPointer
_tmpByte := GetByte();
                
END_METHOD

/// returns a BOOL from the payload buffer from the current payload pointer address and increase the payload pointer afterwards
METHOD GetBool : BOOL
VAR
  /// temporary byte
  _tmpByte : BYTE;
END_VAR
                  // update internal pointer
UpdatePointer();

// check pointer is valid ? 
IF (pPayload = RobotLibraryConstants.NULL_POINTER)
THEN
  RETURN;
END_IF


_tmpByte := GetByte();

// copy data
GetBool := _tmpByte.0;

                
END_METHOD

/// returns a BYTE from the payload buffer from the current payload pointer address and increase the payload pointer afterwards
METHOD GetByte : BYTE
VAR
  /// internal pointer to byte
  _tmpPointer : POINTER TO BYTE;
END_VAR
                  // update internal pointer
UpdatePointer();

// check pointer is valid ? 
IF (pPayload = RobotLibraryConstants.NULL_POINTER)
THEN
  RETURN;
END_IF


_tmpPointer := pPayload + DINT_TO_DWORD(PayloadPtr);

// copy data
GetByte := _tmpPointer^;
// inc payload pointer 
PayloadPtr := PayloadPtr + SIZEOF(BYTE);
                
END_METHOD

/// returns a datablock from the payload buffer from the current payload pointer address and increase the payload pointer afterwards
METHOD GetDataBlock
VAR_INPUT
  /// Target
  pData    : POINTER TO BYTE;
  /// Size of data block
  Size     : UDINT;
  /// Target data type is string ? 
  IsString : BOOL;
END_VAR
                  // update internal pointer
UpdatePointer();

// check pointer is valid ? 
IF (pPayload = RobotLibraryConstants.NULL_POINTER)
THEN
  RETURN;
END_IF


IF ( pData <> RobotLibraryConstants.NULL_POINTER)
THEN
  IF ( IsString)
  THEN
    Size := Size -1;
  END_IF

  // copy data
  SysDepMemCpy(pDest := pData, pSrc := pPayload + DINT_TO_DWORD(PayloadPtr), DataLen := Size);
  
  // inc payload pointer 
  PayloadPtr := PayloadPtr + UDINT_TO_DINT(Size);
END_IF
                
END_METHOD

/// returns a DataInSync from the payload buffer from the current payload pointer address and increase the payload pointer afterwards
METHOD GetDataInSync : DataInSync
VAR
  /// temporary byte
 _tmpByte : BYTE;
END_VAR
                  // update internal pointer
UpdatePointer();

// check pointer is valid ? 
IF (pPayload = RobotLibraryConstants.NULL_POINTER)
THEN
  RETURN;
END_IF


// copy data
_tmpByte := GetByte();

GetDataInSync.ToolsInSync             := _tmpByte.0;
GetDataInSync.FramesInSync            := _tmpByte.1;
GetDataInSync.LoadsInSync             := _tmpByte.2;
GetDataInSync.WorkAreasInSync         := _tmpByte.3;
GetDataInSync.SoftwareLimitsInSync    := _tmpByte.4;
GetDataInSync.DefaultDynamicsInSync   := _tmpByte.5;
GetDataInSync.ReferenceDynamicsInSync := _tmpByte.6;
                
END_METHOD

/// returns a DWORD from the payload buffer from the current payload pointer address and increase the payload pointer afterwards
METHOD GetDword : DWORD
                  // update internal pointer
UpdatePointer();

// check pointer is valid ? 
IF (pPayload = RobotLibraryConstants.NULL_POINTER)
THEN
  RETURN;
END_IF

// copy data
SysDepMemCpy(pDest := ADR(GetDword), pSrc := pPayload + DINT_TO_DWORD(PayloadPtr), DataLen := SIZEOF(DWORD));
// inc payload pointer 
PayloadPtr := PayloadPtr + SIZEOF(DWORD);
                
END_METHOD

/// returns a FragmentAction from the payload buffer from the current payload pointer address and increase the payload pointer afterwards
METHOD GetFragmentAction : FragmentAction
VAR
  /// temporary byte
 _tmpByte : BYTE;
END_VAR
                  // update internal pointer
UpdatePointer();

// check pointer is valid ? 
IF (pPayload = RobotLibraryConstants.NULL_POINTER)
THEN
  RETURN;
END_IF

// copy data
_tmpByte := GetByte();

GetFragmentAction.Complete := _tmpByte.0;
GetFragmentAction.Reset    := _tmpByte.1;
GetFragmentAction.Clear    := _tmpByte.2;
GetFragmentAction.BIT03    := _tmpByte.3;
GetFragmentAction.BIT04    := _tmpByte.4;
GetFragmentAction.BIT05    := _tmpByte.5;
GetFragmentAction.BIT06    := _tmpByte.6;
GetFragmentAction.BIT07    := _tmpByte.7;

                
END_METHOD

/// returns the 1st halfe BYTE from the payload buffer from the current payload pointer address and increase the payload pointer afterwards
METHOD GetHalfeByte1 : BYTE
VAR_INPUT
  /// Increase payload pointer 
  IncPayloadPtr : BOOL;
END_VAR

VAR
  /// temporary byte
 _tmpByte    : BYTE;
  /// internal pointer to byte
 _tmpPointer : POINTER TO BYTE;
END_VAR
                  // update internal pointer
UpdatePointer();

// check pointer is valid ? 
IF (pPayload = RobotLibraryConstants.NULL_POINTER)
THEN
  RETURN;
END_IF

// set pointer
_tmpPointer := pPayload + DINT_TO_DWORD(PayloadPtr); 
// copy data
_tmpByte := _tmpPointer^;

GetHalfeByte1.0 := _tmpByte.0;
GetHalfeByte1.1 := _tmpByte.1;
GetHalfeByte1.2 := _tmpByte.2;
GetHalfeByte1.3 := _tmpByte.3;

IF (IncPayloadPtr)
THEN  
  // inc payload pointer
  PayloadPtr := PayloadPtr + SIZEOF(BYTE);
END_IF
                
END_METHOD

/// returns the 1st halfe BYTE from the payload buffer from the current payload pointer address and increase the payload pointer afterwards
METHOD GetHalfeByte2 : BYTE
VAR_INPUT
  /// Increase payload pointer 
  IncPayloadPtr : BOOL;
END_VAR

VAR
  /// temporary byte
 _tmpByte    : BYTE;
  /// internal pointer to byte
 _tmpPointer : POINTER TO BYTE;
END_VAR
                  // update internal pointer
UpdatePointer();

// check pointer is valid ? 
IF (pPayload = RobotLibraryConstants.NULL_POINTER)
THEN
  RETURN;
END_IF

// set pointer
_tmpPointer := pPayload + DINT_TO_DWORD(PayloadPtr); 
// copy data
_tmpByte := _tmpPointer^;

GetHalfeByte2.0 := _tmpByte.4;
GetHalfeByte2.1 := _tmpByte.5;
GetHalfeByte2.2 := _tmpByte.6;
GetHalfeByte2.3 := _tmpByte.7;

IF (IncPayloadPtr)
THEN  
  // inc payload pointer
  PayloadPtr := PayloadPtr + SIZEOF(BYTE);
END_IF

                
END_METHOD

/// returns a IEC_Date from the payload buffer from the current payload pointer address and increase the payload pointer afterwards
METHOD GetIecDate : IEC_Date
                  // update internal pointer
UpdatePointer();

// check pointer is valid ? 
IF (pPayload = RobotLibraryConstants.NULL_POINTER)
THEN
  RETURN;
END_IF

// copy data
SysDepMemCpy(pDest := ADR(GetIecDate), pSrc := pPayload + DINT_TO_DWORD(PayloadPtr), DataLen := SIZEOF(IEC_DATE));
// swap byte order
GetIecDate := SwapIecDate(GetIecDate);
// inc payload pointer   
PayloadPtr := PayloadPtr + SIZEOF(IEC_DATE);
                
END_METHOD

/// returns a IEC_TIME from the payload buffer from the current payload pointer address and increase the payload pointer afterwards
METHOD GetIecTime : IEC_TIME
                  // update internal pointer
UpdatePointer();

// check pointer is valid ? 
IF (pPayload = RobotLibraryConstants.NULL_POINTER)
THEN
  RETURN;
END_IF

// copy data
SysDepMemCpy(pDest := ADR(GetIecTime), pSrc := pPayload + DINT_TO_DWORD(PayloadPtr), DataLen := SIZEOF(IEC_TIME));
// swap byte order
GetIecTime := SwapIecTime(GetIecTime);
// inc payload pointer   
PayloadPtr := PayloadPtr + SIZEOF(IEC_TIME);
                
END_METHOD

/// returns a INT from the payload buffer from the current payload pointer address and increase the payload pointer afterwards
METHOD GetInt : INT
                  // update internal pointer
UpdatePointer();

// check pointer is valid ? 
IF (pPayload = RobotLibraryConstants.NULL_POINTER)
THEN
  RETURN;
END_IF

// copy data
SysDepMemCpy(pDest := ADR(GetInt), pSrc := pPayload + DINT_TO_DWORD(PayloadPtr), DataLen := SIZEOF(INT));
// swap byte order
GetInt := SwapInt(GetInt);
// inc payload pointer   
PayloadPtr := PayloadPtr + SIZEOF(INT);
                
END_METHOD

/// returns a REAL from the payload buffer from the current payload pointer address and increase the payload pointer afterwards
METHOD GetReal : REAL
                  // update internal pointer
UpdatePointer();

// check pointer is valid ? 
IF (pPayload = RobotLibraryConstants.NULL_POINTER)
THEN
  RETURN;
END_IF

// copy data
SysDepMemCpy(pDest := ADR(GetReal), pSrc := pPayload + DINT_TO_DWORD(PayloadPtr), DataLen := SIZEOF(REAL));
// swap byte order
GetReal := SwapReal(GetReal);
// inc payload pointer   
PayloadPtr := PayloadPtr + SIZEOF(Real);
                
END_METHOD

/// returns a SINT from the payload buffer from the current payload pointer address and increase the payload pointer afterwards
METHOD GetSint : SINT
                  // update internal pointer
UpdatePointer();

// check pointer is valid ? 
IF (pPayload = RobotLibraryConstants.NULL_POINTER)
THEN
  RETURN;
END_IF

// copy data
SysDepMemCpy(pDest := ADR(GetSint), pSrc := pPayload + DINT_TO_DWORD(PayloadPtr), DataLen := SIZEOF(SINT));
// inc payload pointer 
PayloadPtr := PayloadPtr + SIZEOF(SINT);
                
END_METHOD

/// returns a String from the payload buffer from the current payload pointer address and increase the payload pointer afterwards
METHOD GetString : STRING(255)
VAR_INPUT
  Size : DINT;
END_VAR
                  // update internal pointer
UpdatePointer();

// check pointer is valid ? 
IF (pPayload = RobotLibraryConstants.NULL_POINTER)
THEN
  RETURN;
END_IF

// copy data
SysDepMemCpy(pDest := ADR(GetString), pSrc := pPayload + DINT_TO_DWORD(PayloadPtr), DataLen := DINT_TO_UDINT(Size));

// inc payload pointer 
PayloadPtr := PayloadPtr + Size;
                
END_METHOD

/// returns a TrackingStatus from the payload buffer from the current payload pointer address and increase the payload pointer afterwards
METHOD GetTrackingStatus : TrackingStatus
VAR
  /// temporary byte
  tmpByte : BYTE;
END_VAR
                  // update internal pointer
UpdatePointer();

// check pointer is valid ? 
IF (pPayload = RobotLibraryConstants.NULL_POINTER)
THEN
  RETURN;
END_IF

// copy data
tmpByte := GetByte();

GetTrackingStatus.ConveyorTrackingEnabled   := tmpByte.0;  
GetTrackingStatus.WaitingForSynchronization := tmpByte.1;
GetTrackingStatus.Synchronizing             := tmpByte.2;
GetTrackingStatus.Synchronous               := tmpByte.3;
GetTrackingStatus.Desynchronizing           := tmpByte.4;
GetTrackingStatus.SyncOutZoneEntered        := tmpByte.5;
GetTrackingStatus.SyncOutZoneLeft           := tmpByte.6;
GetTrackingStatus.NotUsed                   := tmpByte.7;   
                
END_METHOD

/// returns a TurnNumber from the payload buffer from the current payload pointer address and increase the payload pointer afterwards
METHOD GetTurnNumbers : TurnNumber
                  // update internal pointer
UpdatePointer();

// check pointer is valid ? 
IF (pPayload = RobotLibraryConstants.NULL_POINTER)
THEN
  RETURN;
END_IF

GetTurnNumbers.J1Turns := BYTE_TO_SINT(GetHalfeByte1(FALSE));
GetTurnNumbers.J2Turns := BYTE_TO_SINT(GetHalfeByte2(TRUE));

GetTurnNumbers.J3Turns := BYTE_TO_SINT(GetHalfeByte1(FALSE));
GetTurnNumbers.J4Turns := BYTE_TO_SINT(GetHalfeByte2(TRUE));

GetTurnNumbers.J5Turns := BYTE_TO_SINT(GetHalfeByte1(FALSE));
GetTurnNumbers.J6Turns := BYTE_TO_SINT(GetHalfeByte2(TRUE));

GetTurnNumbers.E1Turns := BYTE_TO_SINT(GetByte());
                
END_METHOD

/// returns a UDINT from the payload buffer from the current payload pointer address and increase the payload pointer afterwards
METHOD GetUdint : UDINT
                  // update internal pointer
UpdatePointer();

// check pointer is valid ? 
IF (pPayload = RobotLibraryConstants.NULL_POINTER)
THEN
  RETURN;
END_IF

// copy data
SysDepMemCpy(pDest := ADR(GetUdint), pSrc := pPayload + DINT_TO_DWORD(PayloadPtr), DataLen := SIZEOF(UDINT));
// swap byte order
GetUdint := SwapUdint(GetUdint);
// inc payload pointer   
PayloadPtr := PayloadPtr + SIZEOF(UDINT);
                
END_METHOD

/// returns a UINT from the payload buffer from the current payload pointer address and increase the payload pointer afterwards
METHOD GetUint : UINT
                  // update internal pointer
UpdatePointer();

// check pointer is valid ? 
IF (pPayload = RobotLibraryConstants.NULL_POINTER)
THEN
  RETURN;
END_IF

// copy data
SysDepMemCpy(pDest := ADR(GetUint), pSrc := pPayload + DINT_TO_DWORD(PayloadPtr), DataLen := SIZEOF(UINT));
// swap byte order
GetUint := SwapUint(GetUint);
// inc payload pointer   
PayloadPtr := PayloadPtr + SIZEOF(UINT);
                
END_METHOD

/// returns a USINT from the payload buffer from the current payload pointer address and increase the payload pointer afterwards
METHOD GetUsint : USINT
                  // update internal pointer
UpdatePointer();

// check pointer is valid ? 
IF (pPayload = RobotLibraryConstants.NULL_POINTER)
THEN
  RETURN;
END_IF

// copy data
SysDepMemCpy(pDest := ADR(GetUsint), pSrc := pPayload + DINT_TO_DWORD(PayloadPtr), DataLen := SIZEOF(USINT));
// inc payload pointer 
PayloadPtr := PayloadPtr + SIZEOF(USINT);
                
END_METHOD

/// returns a WORD from the payload buffer from the current payload pointer address and increase the payload pointer afterwards
METHOD GetWord : WORD
                  // update internal pointer
UpdatePointer();

// check pointer is valid ? 
IF (pPayload = RobotLibraryConstants.NULL_POINTER)
THEN
  RETURN;
END_IF

// copy data
SysDepMemCpy(pDest := ADR(GetWord), pSrc := pPayload + DINT_TO_DWORD(PayloadPtr), DataLen := SIZEOF(WORD));
// swap byte order
GetWord := SwapWord(GetWord);
// inc payload pointer   
PayloadPtr := PayloadPtr + SIZEOF(WORD);
                
END_METHOD

/// Resets the payload buffer, the payload pointer and the payload length
METHOD Reset
VAR_INPUT
END_VAR
                  PayloadLen := 0;
PayloadPtr := 0;
                
END_METHOD

METHOD UpdatePointer
VAR_INPUT
END_VAR
                  
                
END_METHOD
END_FUNCTION_BLOCK

{attribute 'pack_mode' := '1'} 
FUNCTION_BLOCK RobotLibraryRecvDataFB EXTENDS RobotLibraryRecvDataBaseFB
// ------------------------------------------------------------------------- 
//  SRCI Robot Library                                                
// ------------------------------------------------------------------------- 
//                                                                           
//  Object:      RobotLibraryRecvDataFB                                       
//  Author:      Thorsten Brach                                                
//  Date:        2024-06-01
//
//  Description:                                              
//   
//                                                                           
//  Copyright: 
//    (C) 2024 Thorsten Brach. All rights reserved                                                                                                                                            
//             Licensed under the MIT License.
//                                                                           
//  Disclaimer:                                                                           
//    This project is provided without any guarantee and can be used for   
//    private and commercial purposes. Any use is at the user’s 
//    own risk and responsibility.
//
// -------------------------------------------------------------------------
VAR_INPUT
  /// Payload
  Payload    : POINTER TO BYTE;
  /// Size of the Payload array
  PayLoadSize : UDINT;
END_VAR

            
          

METHOD GetLifeSignFooter : BYTE
VAR
  /// temporary 
  pLifeSign : POINTER TO BYTE;
END_VAR
                  pLifeSign := Payload + PayLoadSize -1;


GetLifeSignFooter := GetHalfeByteHi(pLifeSign^); 
                
END_METHOD

METHOD UpdatePointer
VAR_INPUT
END_VAR
                  pPayload := Payload;
                
END_METHOD
END_FUNCTION_BLOCK

{attribute 'pack_mode' := '1'} 
FUNCTION_BLOCK RobotLibraryResponseDataFB EXTENDS RobotLibraryRecvDataBaseFB
// ------------------------------------------------------------------------- 
//  SRCI Robot Library                                                
// ------------------------------------------------------------------------- 
//                                                                           
//  Object:      RobotLibraryResponseDataFB                                       
//  Author:      Thorsten Brach                                                
//  Date:        2025-03-29
//
//  Description:                                              
//   
//                                                                           
//  Copyright: 
//    (C) 2025 Thorsten Brach. All rights reserved                                                                                                                                            
//             Licensed under the MIT License.
//                                                                           
//  Disclaimer:                                                                           
//    This project is provided without any guarantee and can be used for   
//    private and commercial purposes. Any use is at the user’s 
//    own risk and responsibility.
//
// -------------------------------------------------------------------------

VAR_INPUT
  /// Payload
  Payload    : ARRAY [0..RobotLibraryParameter.RESPONSE_PAYLOAD_MAX] OF BYTE;
END_VAR

            
          

/// Resets the payload buffer, the payload pointer and the payload length
METHOD Reset
VAR_INPUT
END_VAR
                  SUPER^.Reset();

// Reset payload buffer
SysDepMemSet(pDest := ADR(Payload), Value := 0 , DataLen := SIZEOF(Payload));

                
END_METHOD

METHOD UpdatePointer
VAR_INPUT
END_VAR
                  pPayload := ADR(Payload);
                
END_METHOD

PROPERTY IsPayloadRemaining : BOOL
GET
VAR
END_VAR
                    IsPayloadRemaining := PayloadPtr < UDINT_TO_DINT(PayloadLen );
                  
END_GET
END_PROPERTY
END_FUNCTION_BLOCK

{attribute 'pack_mode' := '1'} 
FUNCTION_BLOCK RobotLibraryCommandDataFB EXTENDS RobotLibrarySendDataBaseFB
// ------------------------------------------------------------------------- 
//  SRCI Robot Library                                                
// ------------------------------------------------------------------------- 
//                                                                           
//  Object:      RobotLibraryCommandDataFB                                      
//  Author:      Thorsten Brach                                                
//  Date:        2025-03-29
//
//  Description:                                              
//    
//                                                                           
//  Copyright: 
//    (C) 2025 Thorsten Brach. All rights reserved                                                                                                                                            
//             Licensed under the MIT License.
//                                                                           
//  Disclaimer:                                                                           
//    This project is provided without any guarantee and can be used for   
//    private and commercial purposes. Any use is at the user’s 
//    own risk and responsibility.
//
// -------------------------------------------------------------------------

VAR_INPUT
  /// Payload
  Payload : ARRAY [0.. RobotLibraryParameter.PARAMETER_PAYLOAD_MAX] OF BYTE;
END_VAR

            
          

/// Resets the payload buffer, the payload pointer and the payload length
METHOD Reset
VAR_INPUT
END_VAR
                  SUPER^.Reset();

// Reset payload buffer
SysDepMemSet(pDest := ADR(Payload), Value := 0 , DataLen := SIZEOF(Payload));
                
END_METHOD

METHOD UpdatePointer
VAR_INPUT
END_VAR
                  pPayload := ADR(Payload);
                
END_METHOD
END_FUNCTION_BLOCK

{attribute 'pack_mode' := '1'} 
FUNCTION_BLOCK RobotLibrarySendDataBaseFB
// ------------------------------------------------------------------------- 
//  SRCI Robot Library                                                
// ------------------------------------------------------------------------- 
//                                                                           
//  Object:      RobotLibrarySendDataFB                                      
//  Author:      Thorsten Brach                                                
//  Date:        2024-06-01
//
//  Description:                                              
//    
//                                                                           
//  Copyright: 
//    (C) 2024 Thorsten Brach. All rights reserved                                                                                                                                            
//             Licensed under the MIT License.
//                                                                           
//  Disclaimer:                                                                           
//    This project is provided without any guarantee and can be used for   
//    private and commercial purposes. Any use is at the user’s 
//    own risk and responsibility.
//
// -------------------------------------------------------------------------
VAR_INPUT
  /// Payload length
  PayloadLen : UDINT;
  /// Payload pointer
  PayloadPtr : UDINT;
END_VAR


VAR
  /// internal pointer to payload 
  pPayload : POINTER TO BYTE;
END_VAR

            
          

/// Adds a ArmConfigParameter to the payload buffer, increase the payload pointer and returns the payload lenght
METHOD AddArmConfig : UDINT
VAR_INPUT
  /// Value to add
  Value : ArmConfigParameter;
END_VAR

VAR
  /// temporary Byte
 _tmpByte : BYTE;
END_VAR
// Table 6-274: "ConfigMode" on "Command Management Layer"
// --------------------------
// --------------------------
// Byte 00 : Bit 00  - Shoulder
//         : Bit 01  - Shoulder
//         : Bit 02  - Shoulder
//         : Bit 03  - Shoulder
//         : Bit 04  - Elbow
//         : Bit 05  - Elbow
//         : Bit 06  - Elbow
//         : Bit 07  - Elbow
// Byte 01 : Bit 00  - Wrist
//         : Bit 01  - Wrist
//         : Bit 02  - Wrist
//         : Bit 03  - Wrist
//         : Bit 04  - Reserve
//         : Bit 05  - Reserve
//         : Bit 06  - Reserve
//         : Bit 07  - Reserve
                  _tmpByte.0 := Value.Shoulder = ArmConfigShoulder.BACK;
_tmpByte.1 := Value.Elbow    = ArmConfigElbow.DOWN;
_tmpByte.2 := Value.Wrist    = ArmConfigWrist.FLIP;

AddByte(_tmpByte);
AddByte(0);

AddArmConfig := PayloadLen; 
                
END_METHOD

/// Adds a BOOL to the payload buffer, increase the payload pointer and returns the payload lenght
METHOD AddBool : UDINT
VAR_INPUT
  /// Value to add
  Value : BOOL;
END_VAR

VAR
  /// temporary byte
 _tmpByte : BYTE := 0;
END_VAR
                  // update internal pointer
UpdatePointer();

// check pointer is valid ? 
IF (pPayload = RobotLibraryConstants.NULL_POINTER)
THEN
  RETURN;
END_IF


_tmpByte.0 := Value;
// copy data 
SysDepMemCpy(pDest := pPayload + PayloadPtr, pSrc := ADR(_tmpByte), DataLen := SIZEOF(_tmpByte));
// inc payload pointer 
PayloadPtr := PayloadPtr + SIZEOF(_tmpByte);
// return payload len
AddBool := PayloadLen := PayloadPtr;
                
END_METHOD

/// Adds a BYTE to the payload buffer, increase the payload pointer and returns the payload lenght
METHOD AddByte : UDINT
VAR_INPUT
  /// Value to add
  Value : BYTE;
END_VAR
                  // update internal pointer
UpdatePointer();

// check pointer is valid ? 
IF (pPayload = RobotLibraryConstants.NULL_POINTER)
THEN
  RETURN;
END_IF


Value := Value;
// copy data 
SysDepMemCpy( pDest := pPayload + PayloadPtr, pSrc := ADR(Value), DataLen := SIZEOF(Value));
// inc payload pointer 
PayloadPtr := PayloadPtr + SIZEOF(Value);
// return payload len
AddByte := PayloadLen := PayloadPtr;
                
END_METHOD

/// Adds a DataBlock to the payload buffer, increase the payload pointer and returns the payload lenght
METHOD AddDataBlock : UDINT
VAR_INPUT
  /// Value to add
  pValue : POINTER TO BYTE;
  /// Size of data block
  Size   : UDINT;
END_VAR
                  // update internal pointer
UpdatePointer();

// check pointer is valid ? 
IF (pPayload = RobotLibraryConstants.NULL_POINTER)
THEN
  RETURN;
END_IF


IF (pValue = 0) OR (Size = 0 )
THEN
  RETURN;
END_IF

// copy data 
SysDepMemCpy( pDest := pPayload + PayloadPtr, pSrc := pValue, DataLen := Size);
// inc payload pointer 
PayloadPtr := PayloadPtr + Size;
// return payload len
AddDataBlock := PayloadLen := PayloadPtr;
                
END_METHOD

/// Adds a DataInSync to the payload buffer, increase the payload pointer and returns the payload lenght
METHOD AddDataEnableSync : UDINT
VAR_INPUT
  /// Value to add
  Value : DataEnableSync;
END_VAR

VAR
  /// temporary Byte
 _tmpByte : BYTE;
END_VAR
                  Value := Value;

_tmpByte.0 := Value.EnableSyncTool;
_tmpByte.1 := Value.EnableSyncFrame;
_tmpByte.2 := Value.EnableSyncLoad;
_tmpByte.3 := Value.EnableSyncWorkArea;
_tmpByte.4 := Value.EnableSyncSWLimits;
_tmpByte.5 := Value.EnableSyncDefaultDynamics;
_tmpByte.6 := Value.EnableSyncReferenceDynamics;


AddByte(_tmpByte);

AddDataEnableSync := PayloadLen; 
                
END_METHOD

/// Adds a DataInSync to the payload buffer, increase the payload pointer and returns the payload lenght
METHOD AddDataInSync : UDINT
VAR_INPUT
  /// Value to add
  Value : DataInSync;
END_VAR

VAR
  /// temporary Byte
 _tmpByte : BYTE;
END_VAR
                  Value := Value;

_tmpByte.0 := Value.ToolsInSync;
_tmpByte.1 := Value.FramesInSync;
_tmpByte.2 := Value.LoadsInSync;
_tmpByte.3 := Value.WorkAreasInSync;
_tmpByte.4 := Value.SoftwareLimitsInSync;
_tmpByte.5 := Value.DefaultDynamicsInSync;
_tmpByte.6 := Value.ReferenceDynamicsInSync;
_tmpByte.7 := FALSE;

AddByte(_tmpByte);

AddDataInSync := PayloadLen; 
                
END_METHOD

/// Adds a DWORD to the payload buffer , increase the payload pointer and returns the payload lenght
METHOD AddDword : UDINT
VAR_INPUT
  /// Value to add
  Value : DWORD;
END_VAR
                  // update internal pointer
UpdatePointer();

// check pointer is valid ? 
IF (pPayload = RobotLibraryConstants.NULL_POINTER)
THEN
  RETURN;
END_IF


// swap byte order
Value := SwapDword(Value);
// copy data 
SysDepMemCpy(pDest := pPayload + PayloadPtr, pSrc := ADR(Value), DataLen := SIZEOF(Value));
// inc data index 
PayloadPtr := PayloadPtr + SIZEOF(Value);
// return payload len
AddDword := PayloadLen := PayloadPtr;
                
END_METHOD

/// Adds two halfe BYTE to the payload buffer , increase the payload pointer and returns the payload lenght
METHOD AddHalfBytes : UDINT
VAR_INPUT
  /// Value to add
  HalfByteHi : BYTE;
  /// Value to add
  HalfByteLo : BYTE;
END_VAR

VAR
  /// internal value
 _value : BYTE;
END_VAR
                  // update internal pointer
UpdatePointer();

// check pointer is valid ? 
IF (pPayload = RobotLibraryConstants.NULL_POINTER)
THEN
  RETURN;
END_IF


_value := CombineHalfBytes( HalfByteHi := HalfByteHi, HalfByteLo := HalfByteLo);
// copy data 
SysDepMemCpy(pDest := pPayload + PayloadPtr, pSrc := ADR(_value), DataLen := SIZEOF(_value));
// inc payload pointer 
PayloadPtr := PayloadPtr + SIZEOF(_value);
// return payload len
AddHalfBytes := PayloadLen := PayloadPtr;
                
END_METHOD

/// Adds a IEC_DATE to the payload buffer, increase the payload pointer and returns the payload lenght
METHOD AddIecDate : UDINT
VAR_INPUT
  /// Value to add
  Value : IEC_DATE;
END_VAR
                  // update internal pointer
UpdatePointer();

// check pointer is valid ? 
IF (pPayload = RobotLibraryConstants.NULL_POINTER)
THEN
  RETURN;
END_IF


Value := SwapIecDate(Value);
// copy data 
SysDepMemCpy(pDest := pPayload + PayloadPtr, pSrc := ADR(Value), DataLen := SIZEOF(Value));
// inc payload pointer 
PayloadPtr := PayloadPtr + SIZEOF(Value);
// return payload len
AddIecDate := PayloadLen := PayloadPtr;
                
END_METHOD

/// Adds a IEC_TIME to the payload buffer, increase the payload pointer and returns the payload lenght
METHOD AddIecTime : UDINT
VAR_INPUT
  /// Value to add
  Value : IEC_TIME;
END_VAR
                  // update internal pointer
UpdatePointer();

// check pointer is valid ? 
IF (pPayload = RobotLibraryConstants.NULL_POINTER)
THEN
  RETURN;
END_IF


Value := SwapIecTime(Value);
// copy data 
SysDepMemCpy(pDest := pPayload + PayloadPtr, pSrc := ADR(Value), DataLen := SIZEOF(Value));
// inc payload pointer 
PayloadPtr := PayloadPtr + SIZEOF(Value);
// return payload len
AddIecTime := PayloadLen := PayloadPtr;
                
END_METHOD

/// Adds a INT to the payload buffer , increase the payload pointer and returns the payload lenght
METHOD AddInt : UDINT
VAR_INPUT
  /// Value to add
  Value : INT;
END_VAR
                  // update internal pointer
UpdatePointer();

// check pointer is valid ? 
IF (pPayload = RobotLibraryConstants.NULL_POINTER)
THEN
  RETURN;
END_IF


// swap byte order
Value := SwapInt(Value);
// copy data 
SysDepMemCpy(pDest := pPayload + PayloadPtr, pSrc := ADR(Value), DataLen := SIZEOF(Value));
// inc data index 
PayloadPtr := PayloadPtr + SIZEOF(Value);
// return payload len
AddInt := PayloadLen := PayloadPtr;
                
END_METHOD

/// Adds a REAL to the payload buffer , increase the payload pointer and returns the payload lenght
METHOD AddReal : UDINT
VAR_INPUT
  /// Value to add
  Value : REAL;
END_VAR
                  // update internal pointer
UpdatePointer();

// check pointer is valid ? 
IF (pPayload = RobotLibraryConstants.NULL_POINTER)
THEN
  RETURN;
END_IF


// swap byte order
Value := SwapReal(Value);
// copy data 
SysDepMemCpy(pDest := pPayload + PayloadPtr,pSrc := ADR(Value), DataLen := SIZEOF(Value));
// inc data index 
PayloadPtr := PayloadPtr + SIZEOF(Value);
// return payload len
AddReal := PayloadLen := PayloadPtr;
                
END_METHOD

/// Adds a SINT to the payload buffer, increase the payload pointer and returns the payload lenght
METHOD AddSint : UDINT
VAR_INPUT
  /// Value to add
  Value : SINT;
END_VAR
                  // update internal pointer
UpdatePointer();

// check pointer is valid ? 
IF (pPayload = RobotLibraryConstants.NULL_POINTER)
THEN
  RETURN;
END_IF


Value := Value;
// copy data 
SysDepMemCpy(pDest := pPayload + PayloadPtr, pSrc := ADR(Value), DataLen := SIZEOF(Value));
// inc payload pointer 
PayloadPtr := PayloadPtr + SIZEOF(Value);
// return payload len
AddSint := PayloadLen := PayloadPtr;
                
END_METHOD

/// Adds a String to the payload buffer, increase the payload pointer and returns the payload lenght
METHOD AddString : UDINT
VAR_INPUT
  /// Value to add
  Value : STRING(255);
END_VAR
                  // update internal pointer
UpdatePointer();

// check pointer is valid ? 
IF (pPayload = RobotLibraryConstants.NULL_POINTER)
THEN
  RETURN;
END_IF


IF ( LEN(Value) = 0 )
THEN
  RETURN;
END_IF

// copy data 
SysDepMemCpy(pDest := pPayload + PayloadPtr, pSrc := ADR(Value), DataLen := DINT_TO_UDINT(LEN(Value)));
// inc payload pointer 
PayloadPtr := PayloadPtr + DINT_TO_UDINT(LEN(Value));
// return payload len
AddString := PayloadLen := PayloadPtr;
                
END_METHOD

/// Adds a TIME to the payload buffer , increase the payload pointer and returns the payload lenght
METHOD AddTime : UDINT
VAR_INPUT
  /// Value to add
  Value : TOD;
END_VAR
                  // update internal pointer
UpdatePointer();

// check pointer is valid ? 
IF (pPayload = RobotLibraryConstants.NULL_POINTER)
THEN
  RETURN;
END_IF


// swap byte order
Value := SwapIecTime(Value);
// copy data 
SysDepMemCpy(pDest := pPayload + PayloadPtr, pSrc := ADR(Value), DataLen := SIZEOF(Value));
// inc data index 
PayloadPtr := PayloadPtr + SIZEOF(Value);
// return payload len
AddTime := PayloadLen := PayloadPtr;
                
END_METHOD

/// Adds a TurnNumber to the payload buffer, increase the payload pointer and returns the payload lenght
METHOD AddTurnNumber : UDINT
VAR_INPUT
  /// Value to add
  Value : TurnNumber;
END_VAR

VAR
  /// temporary Byte
 _tmpByte : BYTE;
END_VAR
                  Value := Value;

AddHalfBytes( HalfByteHi := SINT_TO_BYTE(Value.J2Turns) , HalfByteLo := SINT_TO_BYTE(Value.J1Turns));
AddHalfBytes( HalfByteHi := SINT_TO_BYTE(Value.J4Turns) , HalfByteLo := SINT_TO_BYTE(Value.J3Turns));
AddHalfBytes( HalfByteHi := SINT_TO_BYTE(Value.J6Turns) , HalfByteLo := SINT_TO_BYTE(Value.J5Turns));
AddByte(SINT_TO_BYTE(Value.E1Turns));

AddTurnNumber := PayloadLen; 

                
END_METHOD

/// Adds a UDINT to the payload buffer , increase the payload pointer and returns the payload lenght
METHOD AddUdint : UDINT
VAR_INPUT
  /// Value to add
  Value : UDINT;
END_VAR
                  // update internal pointer
UpdatePointer();

// check pointer is valid ? 
IF (pPayload = RobotLibraryConstants.NULL_POINTER)
THEN
  RETURN;
END_IF


// swap byte order
Value := SwapUdint(Value);
// copy data 
SysDepMemCpy(pDest := pPayload + PayloadPtr, pSrc := ADR(Value), DataLen := SIZEOF(Value));
// inc data index 
PayloadPtr := PayloadPtr + SIZEOF(Value);
// return payload len
AddUdint := PayloadLen := PayloadPtr;
                
END_METHOD

/// Adds a UINT to the payload buffer , increase the payload pointer and returns the payload lenght
METHOD AddUint : UDINT
VAR_INPUT
  /// Value to add
  Value : UINT;
END_VAR
                  // update internal pointer
UpdatePointer();

// check pointer is valid ? 
IF (pPayload = RobotLibraryConstants.NULL_POINTER)
THEN
  RETURN;
END_IF


// swap byte order
Value := SwapUint(Value);
// copy data 
SysDepMemCpy(pDest := pPayload + PayloadPtr, pSrc := ADR(Value), DataLen := SIZEOF(Value));
// inc data index 
PayloadPtr := PayloadPtr + SIZEOF(Value);
// return payload len
AddUint := PayloadLen := PayloadPtr;
                
END_METHOD

/// Adds a USINT to the payload buffer, increase the payload pointer and returns the payload lenght
METHOD AddUsint : UDINT
VAR_INPUT
  /// Value to add
  Value : USINT;
END_VAR
                  // update internal pointer
UpdatePointer();

// check pointer is valid ? 
IF (pPayload = RobotLibraryConstants.NULL_POINTER)
THEN
  RETURN;
END_IF


Value := Value;
// copy data 
SysDepMemCpy(pDest := pPayload + PayloadPtr, pSrc := ADR(Value), DataLen := SIZEOF(Value));
// inc payload pointer 
PayloadPtr := PayloadPtr + SIZEOF(Value);
// return payload len
AddUsint := PayloadLen := PayloadPtr;
                
END_METHOD

/// Resets the payload buffer, the payload pointer and the payload length
METHOD Reset
VAR_INPUT
END_VAR
                  PayloadLen := 0;
PayloadPtr := 0;
                
END_METHOD

METHOD UpdatePointer
VAR_INPUT
END_VAR
                  
                
END_METHOD
END_FUNCTION_BLOCK

{attribute 'pack_mode' := '1'} 
FUNCTION_BLOCK RobotLibrarySendDataFB extends RobotLibrarySendDataBaseFB
// ------------------------------------------------------------------------- 
//  SRCI Robot Library                                                
// ------------------------------------------------------------------------- 
//                                                                           
//  Object:      RobotLibrarySendDataFB                                      
//  Author:      Thorsten Brach                                                
//  Date:        2024-06-01
//
//  Description:                                              
//    
//                                                                           
//  Copyright: 
//    (C) 2024 Thorsten Brach. All rights reserved                                                                                                                                            
//             Licensed under the MIT License.
//                                                                           
//  Disclaimer:                                                                           
//    This project is provided without any guarantee and can be used for   
//    private and commercial purposes. Any use is at the user’s 
//    own risk and responsibility.
//
// -------------------------------------------------------------------------
VAR_INPUT
  /// Payload
  Payload     : POINTER TO BYTE;
  /// Size of the Payload array
  PayLoadSize : UDINT;
END_VAR

            
          

/// Resets the payload buffer, the payload pointer and the payload length
METHOD Reset
VAR_INPUT
END_VAR
                  SUPER^.Reset();

// Reset payload buffer
SysDepMemSet(pDest := Payload, Value := 0 , DataLen := PayLoadSize);
                
END_METHOD

METHOD SetLifeSignFooter
VAR_INPUT
  /// Life sign value
  LifeSign : BYTE;
END_VAR

VAR
  /// temporary 
  pLifeSign : POINTER TO BYTE;
END_VAR
                  pLifeSign := Payload + PayLoadSize -1;

pLifeSign^ := LifeSign;
                
END_METHOD

METHOD UpdatePointer
VAR_INPUT
END_VAR
                  pPayload := Payload;
                
END_METHOD
END_FUNCTION_BLOCK

FUNCTION_BLOCK AxesGroupSystemDataFB 
{attribute 'pack_mode' := '1'} 
// ------------------------------------------------------------------------- 
//  SRCI Robot Library                                                
// ------------------------------------------------------------------------- 
//                                                                           
//  Object:      AxesGroupSystemDataFB                                       
//  Author:      Thorsten Brach                                                
//  Date:        2025-08-31
//
//  Description:                                              
//   
//                                                                           
//  Copyright: 
//    (C) 2025 Thorsten Brach. All rights reserved                                                                                                                                            
//             Licensed under the MIT License.
//                                                                           
//  Disclaimer:                                                                           
//    This project is provided without any guarantee and can be used for   
//    private and commercial purposes. Any use is at the user’s 
//    own risk and responsibility.
//
// -------------------------------------------------------------------------
VAR_INPUT
  /// Pointer to ToolData array
  ToolDataPtr       : POINTER TO Tool;
  /// Lower dimension of ToolData array 
  ToolDataMin       : DINT;
  /// Lower dimension of ToolData array
  ToolDataMax       : DINT;
  /// Amount of ToolData elements in array
  ToolDataCount     : UDINT;

  /// Pointer to LoadData array
  LoadDataPtr       : POINTER TO Load;
  /// Lower dimension of LoadData array 
  LoadDataMin       : DINT;
  /// Lower dimension of LoadData array
  LoadDataMax       : DINT;
  /// Amount of Load elements in array
  LoadDataCount     : UDINT;

  /// Pointer to FrameData array
  FrameDataPtr      : POINTER TO Frame;
  /// Lower dimension of FrameData array 
  FrameDataMin      : DINT;
  /// Lower dimension of FrameData array
  FrameDataMax      : DINT;
  /// Amount of FrameData elements in array
  FrameDataCount    : UDINT;
  
  /// Pointer to WorkAreas array
  WorkAreasPtr      : POINTER TO RobotWorkArea;
  /// Lower dimension of WorkAreas array 
  WorkAreasMin      : DINT;
  /// Lower dimension of WorkAreas array
  WorkAreasMax      : DINT;
  /// Amount of WorkAreas elements in array
  WorkAreasCount    : UDINT;
  
  /// Software limits stored on PLC
  SWLimits          : REFERENCE TO SWLimits;
  /// Default dynamics stored on PLC. For more information refer to 5.5.7
  DefaultDynamics   : REFERENCE TO DefaultDynamics;
  /// Reference dynamics stored on PLC. For more information refer to 5.5.7
  ReferenceDynamics : REFERENCE TO ReferenceDynamics;
END_VAR

            
          

METHOD UpdateDefaultDynamics : DINT
VAR_INPUT
  /// Default dynamics values according to Table 6-148.
  DynamicValues : DefaultDynamics;
END_VAR
                  // Check pointer is vaild ?
IF ( NOT __ISVALIDREF(DefaultDynamics))  
THEN
  RETURN;
END_IF

// Applay new values
DefaultDynamics := DynamicValues;
                
END_METHOD

METHOD UpdateFrameData : DINT
VAR_INPUT
  /// Reference to BaseFB 
  Caller     : REFERENCE TO RobotLibraryBaseFB;
  /// Current System Time
  SystemTime : SystemTime;
  /// Frame index M
  /// • 0: WCS (default) O
  /// • 1..254: UCS (User frames)
  FrameNo    : USINT;
  /// Frame data (see chapter 5.5.6.2)
  FrameData  : FrameData;
END_VAR


VAR
  /// pointer to frame data
  pFrameData : POINTER TO Frame;  
END_VAR
                  // Check pointer is vaild ?
IF ( FrameDataPtr = RobotLibraryConstants.NULL_POINTER )
THEN
  RETURN;
END_IF

// Check Frame number is in range ?
IF (( FrameNo < FrameDataMin ) OR
    ( FrameNo > FrameDataMax ))
THEN
  IF ( __ISVALIDREF( Caller ))
  THEN
   // set warning
   Caller.SetWarning( WarningID := RobotLibraryWarningIdEnum.WARN_SAVE_FRAME_FAILED, Overwrite := FALSE);
   
   // Create log entry
   Caller.CreateLogMessagePara1 ( Timestamp   := SystemTime,
                                  MessageType := MessageType.CMD,
                                  Severity    := Severity.WARNING,
                                  MessageCode := Caller.WarningID,
                                  MessageText := 'Save FrameData failed. Index {1} not available in user defined system data',
                                  Para1       :=  USINT_TO_STRING(FrameNo));
  END_IF

  RETURN;
END_IF


// Calculate pointer address for the index of the FrameData Array
pFrameData := FrameDataPtr + (( FrameNo - DINT_TO_UDINT(FrameDataMin)) * SIZEOF(Frame));
// copy frame data to Array index
pFrameData^.Available := TRUE;
pFrameData^.Data := FrameData;
                
END_METHOD

METHOD UpdateLoadData : DINT
VAR_INPUT
  /// Reference to BaseFB 
  Caller     : REFERENCE TO RobotLibraryBaseFB;
  /// Current System Time
  SystemTime : SystemTime;
  /// Specifies the desired target values that shall be written
  /// Load index
  /// •      0: (default) - Not possible to write
  /// • 1..254: Load data
  LoadNo     : USINT;
  /// Load data (see chapter 5.5.6.4)
  LoadData   : LoadData;
END_VAR


VAR
  /// pointer to load data
  pLoadData : POINTER TO Load;  
END_VAR
                  // Check pointer is vaild ?
IF ( LoadDataPtr = RobotLibraryConstants.NULL_POINTER )
THEN
  RETURN;
END_IF

// Check Load number is in range ?
IF (( LoadNo < LoadDataMin ) OR
    ( LoadNo > LoadDataMax ))
THEN
  IF ( __ISVALIDREF( Caller ))
  THEN
   // set warning
   Caller.SetWarning( WarningID := RobotLibraryWarningIdEnum.WARN_SAVE_LOAD_FAILED, Overwrite := FALSE);
   
   // Create log entry
   Caller.CreateLogMessagePara1 ( Timestamp   := SystemTime,
                                  MessageType := MessageType.CMD,
                                  Severity    := Severity.WARNING,
                                  MessageCode := Caller.WarningID,
                                  MessageText := 'Save LoadData failed. Index {1} not available in user defined system data',
                                  Para1       :=  USINT_TO_STRING(LoadNo));
  END_IF

  RETURN;
END_IF


// Calculate pointer address for the index of the LoadData Array
pLoadData := LoadDataPtr + (( LoadNo - DINT_TO_UDINT(LoadDataMin)) * SIZEOF(Load));
// copy load data to Array index
pLoadData^.Available := TRUE;
pLoadData^.Data := LoadData;
                
END_METHOD

METHOD UpdateReferenceDynamics : DINT
VAR_INPUT
  /// Reference dynamics values according to Table 6-109.
  DynamicValues : ReferenceDynamics;
END_VAR
                  // Check pointer is vaild ?
IF ( NOT __ISVALIDREF(ReferenceDynamics))  
THEN
  RETURN;
END_IF

// Applay new values
ReferenceDynamics := DynamicValues;
                
END_METHOD

METHOD UpdateSWLimits : DINT
VAR_INPUT
  /// Limits for joints and external axes according to Table 6-180.
  LimitValues : SWLimits;
END_VAR
                  // Check pointer is vaild ?
IF ( NOT __ISVALIDREF(SWLimits))  
THEN
  RETURN;
END_IF

// Applay new values
SWLimits := LimitValues;
                
END_METHOD

METHOD UpdateToolData : DINT
VAR_INPUT
  /// Reference to BaseFB 
  Caller     : REFERENCE TO RobotLibraryBaseFB;
  /// Current System Time
  SystemTime : SystemTime;
  /// Tool index
  /// •      0: Flange (default) Not possible to change
  /// • 1..254: Tool Frame
  ToolNo     : USINT;
  /// Tool data (see chapter 5.5.6.3)
  ToolData   : ToolData;
END_VAR


VAR
  /// pointer to tool data
  pToolData : POINTER TO TOOL;  
END_VAR
                  // Check pointer is vaild ?
IF ( ToolDataPtr = RobotLibraryConstants.NULL_POINTER )
THEN
  RETURN;
END_IF

// Check Tool number is in range ?
IF (( ToolNo < ToolDataMin ) OR
    ( ToolNo > ToolDataMax ))
THEN
  IF ( __ISVALIDREF( Caller ))
  THEN
   // set warning
   Caller.SetWarning( WarningID := RobotLibraryWarningIdEnum.WARN_SAVE_TOOL_FAILED, Overwrite := FALSE);
   
   // Create log entry
   Caller.CreateLogMessagePara1 ( Timestamp   := SystemTime,
                                  MessageType := MessageType.CMD,
                                  Severity    := Severity.WARNING,
                                  MessageCode := Caller.WarningID,
                                  MessageText := 'Save ToolData failed. Index {1} not available in user defined system data',
                                  Para1       :=  USINT_TO_STRING(ToolNo));
  END_IF

  RETURN;
END_IF

{warning 'ToDo: Compiler Fehler'}
(*

// Calculate pointer address for the index of the ToolData Array
pToolData := ToolDataPtr + (( ToolNo - DINT_TO_UDINT(ToolDataMin)) * SIZEOF(Tool));
// copy tool data to Array index
pToolData^.Available := TRUE;
pToolData^.Data := ToolData;

*)

                
END_METHOD

METHOD UpdateWorAreas : DINT
VAR_INPUT
  /// Reference to BaseFB 
  Caller       : REFERENCE TO RobotLibraryBaseFB;
  /// Current System Time
  SystemTime   : SystemTime;
  /// Index of the robot work area
  /// • 0 (default)..254
  WorkAreaNo   : USINT;
  /// Data specific to the work area requested by Index.
  WorkAreaData : RobotWorkAreaData;
END_VAR
VAR
  /// pointer to WorkArea
  pWorkAreaData : POINTER TO RobotWorkArea;  
END_VAR
                  // Check pointer is vaild ?
IF ( WorkAreasPtr = RobotLibraryConstants.NULL_POINTER )
THEN
  RETURN;
END_IF

// Check WorkArea number is in range ?
IF (( WorkAreaNo < WorkAreasMin ) OR
    ( WorkAreaNo > WorkAreasMax ))
THEN
  IF ( __ISVALIDREF( Caller ))
  THEN
   // set warning
   Caller.SetWarning( WarningID := RobotLibraryWarningIdEnum.WARN_SAVE_WORKAREA_FAILED, Overwrite := FALSE);
   
   // Create log entry
   Caller.CreateLogMessagePara1 ( Timestamp   := SystemTime,
                                  MessageType := MessageType.CMD,
                                  Severity    := Severity.WARNING,
                                  MessageCode := Caller.WarningID,
                                  MessageText := 'Save WorkArea failed. Index {1} not available in user defined system data',
                                  Para1       :=  USINT_TO_STRING(WorkAreaNo));
  END_IF

  RETURN;
END_IF


// Calculate pointer address for the index of the WorkArea Array
pWorkAreaData := WorkAreasPtr + (( WorkAreaNo - DINT_TO_UDINT(WorkAreasMin)) * SIZEOF(RobotWorkArea));
// copy WorkArea to Array index
pWorkAreaData^.Available := TRUE;
pWorkAreaData^.Data := WorkAreaData;
                
END_METHOD
END_FUNCTION_BLOCK

FUNCTION_BLOCK ActiveCommandRegisterFB EXTENDS RobotLibraryLogFB
// ------------------------------------------------------------------------- 
//  SRCI Robot Library                                                
// ------------------------------------------------------------------------- 
//                                                                           
//  Object:      ActiveCommandRegisterFB                                       
//  Author:      Thorsten Brach                                                
//  Date:        2024-06-01
//
//  Description:                                              
//   
//                                                                           
//  Copyright: 
//    (C) 2024 Thorsten Brach. All rights reserved                                                                                                                                            
//             Licensed under the MIT License.
//                                                                           
//  Disclaimer:                                                                           
//    This project is provided without any guarantee and can be used for   
//    private and commercial purposes. Any use is at the user’s 
//    own risk and responsibility.
//
// -------------------------------------------------------------------------
VAR_INPUT
  /// Active Command Register
  Register            : ARRAY [1..RobotLibraryParameter.ACTIVE_CMD_REGISTER_ENTRIES_MAX] OF AxesGroupAcyclicAcrEntry;
  /// System Time
  SystemTime          : SystemTime;
  /// usable size of the arc register
  RegisterSize        : DINT := RobotLibraryParameter.ACTIVE_CMD_REGISTER_ENTRIES_MAX;
END_VAR

VAR_OUTPUT
  /// Execution Order List 
  ExecutionOrderList    : ARRAY [1..RobotLibraryParameter.ACTIVE_CMD_REGISTER_ENTRIES_MAX] OF DINT;
  /// Current amount of used registers
  CurrentAcrUsageCount  : DINT;  
  /// Current percent of used registers
  CurrentAcrUsagePercent : REAL;    
END_VAR


VAR
  /// temporarty Active Command Register
  TmpRegister                 : ARRAY [1..RobotLibraryParameter.ACTIVE_CMD_REGISTER_ENTRIES_MAX] OF AxesGroupAcyclicAcrEntry;
  /// last used unique ID 
  LastUniqueID                : UINT;
  /// Warning for ACR usage at 80%
  WarningAcrUsage             : R_TRIG;
END_VAR

VAR CONSTANT
  /// Active command
  ACTIVE_CMD           : UDINT := 1;
  /// Buffered command
  BUFFER_CMD           : UDINT := 2;
  /// Empty ACR entry
  EMPTY_ACR_ENTRY      : AxesGroupAcyclicAcrEntry := (State := ActiveCommandRegisterState.IS_FREE);
  /// Empty command entry
  EMPTY_CMD_ENTRY      : AxesGroupAcyclicAcrEntryCmdBuffer := (State := BufferStateCmd.EMPTY);  
  /// constant for byte index of priority in payload 
  PRIORITY_IDX         : BYTE := 3;  
  /// bitmask to mask the priority out of the halfbyte
  PRIORITY_BIT_MASK    : BYTE := 2#000_1111;   
END_VAR

            ManageRegister();

UpdateExecutionOrderList();
          

METHOD PUBLIC AddCmd : UDINT
VAR_INPUT
  /// Pointer to the corresponding command-FB to enable a callback mechanism
  pCommandFB        : POINTER TO RobotLibraryBaseFB;
END_VAR

VAR
  /// internal index for loops
 _regIdx            : DINT;
  /// internal command type 
 _cmdType           : CmdType;
  /// log message
 _messageLog        : AlarmMessage;  
  /// flag for free register found
 _freeRegisterFound : BOOL;
  /// internal Acr error 
 _errorAcrEntry     : WORD := RobotLibraryErrorIdEnum.ERR_NO_FREE_ACR_ENTRY;  
END_VAR
                  // calculate the used length of the ACR 
FOR _regIdx := 1 TO RegisterSize
DO
  IF ( Register[_regIdx].State = ActiveCommandRegisterState.IS_FREE )
  THEN
    Register[_regIdx].State      := ActiveCommandRegisterState.IS_PROCESSING;
    Register[_regIdx].UniqueID   := DINT_TO_UINT(_regIdx);
    Register[_regIdx].pCommandFB := pCommandFB;

    // check pointer to command FB
    IF ( Register[_regIdx].pCommandFB <> RobotLibraryConstants.NULL_POINTER )
    THEN
      Register[_regIdx].Command[RobotLibraryConstants.ACTIVE_CMD].Timestamp  := SystemTime;

      Register[_regIdx].Command[RobotLibraryConstants.ACTIVE_CMD].Payload    := pCommandFB^.CommandData.Payload; 
      Register[_regIdx].Command[RobotLibraryConstants.ACTIVE_CMD].PayloadLen := pCommandFB^.CommandData.PayloadLen;
      Register[_regIdx].Command[RobotLibraryConstants.ACTIVE_CMD].PayLoadPtr := 0;
      Register[_regIdx].Command[RobotLibraryConstants.ACTIVE_CMD].State      := BufferStateCmd.CREATED;
    END_IF
  
    // set flag for free register found
   _freeRegisterFound := TRUE;
    
    // Increment Current used register counter
    CurrentAcrUsageCount := CurrentAcrUsageCount + 1;
    
    // return Unique ID
    AddCmd := Register[_regIdx].UniqueID;

    // Get CmdType from payload
    SysDepMemCpy( pDest := ADR(_cmdType), pSrc := ADR(pCommandFB^.CommandData.Payload), DataLen := SIZEOF(_cmdType));
    
    // Create log entry
    CreateLogMessagePara2 ( Timestamp   := SystemTime,
                            MessageType := MessageType.CMD,
                            Severity    := Severity.INFO,
                            MessageCode := 0,
                            MessageText := 'ACR-ID [{1}]: Added  Command-Payload of CmdType <{2}>',
                            Para1       :=  DINT_TO_STRING(_regIdx),
                            Para2       :=  CMD_TYPE_TO_STRING(SwapUint(_cmdType)));
    EXIT;
  END_IF
END_FOR

// Check a free register could be found ? 
IF ( NOT _freeRegisterFound )
THEN
  // set error in Command FB   
  IF ( pCommandFB <> RobotLibraryConstants.NULL_POINTER )
  THEN
    SysDepMemCpy( pDest   := ADR   ( pCommandFB^.ErrorID ), 
                  pSrc    := ADR   ( _errorAcrEntry      ),
                  DataLen := SIZEOF( _errorAcrEntry      )); 
  END_IF


  // Create log entry
  CreateLogMessagePara1 ( Timestamp   := SystemTime,
                          MessageType := MessageType.CMD,
                          Severity    := Severity.FATAL_ERROR,
                          MessageCode := 0,
                          MessageText := 'Not possible to add CMD <{1}> to ACR - NO FREE REGISTER FOUND ! -> STOPPING SRCI INTERFACE...',
                          Para1       :=  CMD_TYPE_TO_STRING(SwapUint(_cmdType)));                          
END_IF
                
END_METHOD

METHOD AddRsp : UDINT
VAR_INPUT
  /// Response
  Rsp : TelegramRobToPlcFragment;
END_VAR
VAR
  /// internal index for loops
 _Idx             : DINT;
  /// internal registen index
 _regIdx          : DINT;
  /// internal command type
 _cmdType         : CmdType;
  /// internal FragmentAction
 _fragmentAction  :  FragmentAction;
  /// internal command message state
 _cmdMessageState : CmdMessageState;
  /// internal flag for CmdID found
 _found           : BOOL;
END_VAR
                  FOR _regIdx := 1 TO RegisterSize
DO
  IF ( Register[_regIdx].UniqueID = Rsp.Header.CmdID )
  THEN
    // CmdID was found in the ACR
   _found := TRUE;
    // convert to fragment action 
   _fragmentAction := ByteToFragmentAction(Rsp.Header.FragmentAction);

    // delete response 
    IF ( _fragmentAction.Clear )
    THEN
      SysDepMemSet( pDest := ADR(Register[_regIdx].Response[ACTIVE_CMD]), Value := 0, DataLen := SIZEOF(Register[_regIdx].Response[ACTIVE_CMD]));
    END_IF
                       
    // add payload to response
    FOR _idx := Rsp.Header.PayloadPointer TO  Rsp.Header.PayloadLength -1
    DO
      Register[_regIdx].Response[ACTIVE_CMD].Timestamp     := SystemTime;
      Register[_regIdx].Response[ACTIVE_CMD].State         := BufferStateRsp.RECEIVING;
      Register[_regIdx].Response[ACTIVE_CMD].PayloadLen    := Register[_regIdx].Response[ACTIVE_CMD].PayloadLen + 1;
      Register[_regIdx].Response[ACTIVE_CMD].Payload[_idx] := Rsp.Command.Payload[_idx];
    END_FOR

    // Get current message state 
   _cmdMessageState := GetHalfeByteLo    (Value  := Register[_regIdx].Response[ACTIVE_CMD].Payload[0]);
    // Get command type from payload
   _cmdType         := CombineBytesToUint(HiByte := Register[_regIdx].Command [ACTIVE_CMD].Payload[0],
                                          LoByte := Register[_regIdx].Command [ACTIVE_CMD].Payload[1]);

    // Create log entry
    CreateLogMessagePara3 ( Timestamp   := SystemTime,
                            MessageType := MessageType.CMD,
                            Severity    := Severity.INFO,
                            MessageCode := 0,
                            MessageText := 'ACR-ID [{1}]: Added Response-Payload of CmdType <{2}> with State = {3}',
                            Para1       :=  DINT_TO_STRING(_regIdx),
                            Para2       :=  CMD_TYPE_TO_STRING(_cmdType),
                            Para3       :=  CMD_MESSAGE_STATE_TO_STRING(_cmdMessageState));

    IF ( _fragmentAction.Complete )
    THEN
      // set response state
      Register[_regIdx].Response[ACTIVE_CMD].State := BufferStateRsp.RECEIVED;      
     
      // Check current message state and tag the register state as IS_FINAL, if needed 
      IF ( _cmdMessageState >= CmdMessageState.DONE) 
      THEN
        Register[_regIdx].State := ActiveCommandRegisterState.IS_FINAL;
        
        // get command type from payload
       _cmdType := CombineBytesToUint(HiByte := Register[_regIdx].Command[ACTIVE_CMD].Payload[0],
                                      LoByte := Register[_regIdx].Command[ACTIVE_CMD].Payload[1]);

        // Create log entry
        CreateLogMessagePara3( Timestamp   := SystemTime,
                               MessageType := MessageType.CMD,
                               Severity    := Severity.INFO,
                               MessageCode := 0,
                               MessageText := 'ACR-ID [{1}]: Detected Response-Payload of CmdType <{2}> has reached final state <{3}>',
                               Para1       :=  DINT_TO_STRING(_regIdx),
                               Para2       :=  CMD_TYPE_TO_STRING(_cmdType),
                               Para3       :=  CMD_MESSAGE_STATE_TO_STRING(_cmdMessageState));
                               
        // Exit the loop
      END_IF      
    END_IF
    
    
    // Check Response received complete ? 
    IF ( Register[_regIdx].Response[ACTIVE_CMD].State = BufferStateRsp.RECEIVED)
    THEN
      // update state
      Register[_regIdx].Response[ACTIVE_CMD].State := BufferStateRsp.PROCESSED;
      // callback CommandFB    
      Register[_regIdx].pCommandFB^.CallBack(RspData := Register[_regIdx].Response[ACTIVE_CMD],TimeStamp := SystemTime);    
    END_IF
    
    EXIT;
  END_IF
END_FOR


// Check CmdID was found in the ACR ? 
IF ( NOT _found )
THEN
  // Create log entry
  CreateLogMessagePara2 ( Timestamp   := SystemTime,
                          MessageType := MessageType.CMD,
                          Severity    := Severity.WARNING,
                          MessageCode := 0,
                          MessageText := 'ACR-ID [?]: Response-Payload of CmdID <{1}> with State = {2} received, but no matching ACR entry found',
                          Para1       :=  UINT_TO_STRING(Rsp.Header.CmdID),
                          Para2       :=  CMD_MESSAGE_STATE_TO_STRING(_cmdMessageState));
END_IF
                
END_METHOD

METHOD FB_init : BOOL
VAR_INPUT
  bInitRetains : BOOL; // if TRUE, the retain variables are initialized (warm start / cold start)
  bInCopyCode : BOOL;  // if TRUE, the instance afterwards gets moved into the copy code (online change)
END_VAR
                  MyType := 'ActiveCommandRegisterFB';


                
END_METHOD

METHOD PRIVATE ManageRegister
VAR
  /// internal index
 _regIdx          : DINT;
  /// internal command type
 _cmdType         : CmdType;
  /// internal command message state
 _cmdMessageState : CmdMessageState; 
END_VAR
                  FOR _regIdx := 1 TO RegisterSize
DO
  // Check pointer to command FB is valid ? 
  IF ( Register[_regIdx].pCommandFB <> RobotLibraryConstants.NULL_POINTER) 
  THEN
  
    // Check apply Cmd parameter update ?  
    IF (( Register[_regIdx].Command[ACTIVE_CMD].State = BufferStateCmd.PROCESSED        ) AND
        ( Register[_regIdx].Command[BUFFER_CMD].State = BufferStateCmd.UPDATE_AVAILABLE ))
    THEN
      Register[_regIdx].Command[ACTIVE_CMD] := Register[_regIdx].Command[BUFFER_CMD];
      Register[_regIdx].Command[BUFFER_CMD] := EMPTY_CMD_ENTRY;
  
      // get command type from payload
     _cmdType := CombineBytesToUint(HiByte := Register[_regIdx].Command[ACTIVE_CMD].Payload[0],
                                    LoByte := Register[_regIdx].Command[ACTIVE_CMD].Payload[1]);
  
      // Create log entry
      CreateLogMessagePara2 ( Timestamp   := SystemTime,
                              MessageType := MessageType.CMD,
                              Severity    := Severity.INFO,
                              MessageCode := 0,
                              MessageText := 'ACR-ID [{1}]: Moved BUFFER_CMD to ACTIVE_CMD, CmdType <{2}>',
                              Para1       :=  DINT_TO_STRING(_regIdx),
                              Para2       :=  CMD_TYPE_TO_STRING(_cmdType));
  
    END_IF
    
    (*
    // Check Response received ? 
    IF ( Register[_regIdx].Response[ACTIVE_CMD].State = BufferStateRsp.RECEIVED)
    THEN
      // update state
      Register[_regIdx].Response[ACTIVE_CMD].State := BufferStateRsp.PROCESSED;
      // callback CommandFB    
      Register[_regIdx].pCommandFB^.CallBack(RspData := Register[_regIdx].Response[ACTIVE_CMD],TimeStamp := SystemTime);    
    END_IF
    *)
    
    // delete entries with State.IS_Final 
    IF ( Register[_regIdx].State = ActiveCommandRegisterState.IS_FINAL )
    THEN
      // get command type from payload
     _cmdType := CombineBytesToUint(HiByte := Register[_regIdx].Command[ACTIVE_CMD].Payload[0],
                                    LoByte := Register[_regIdx].Command[ACTIVE_CMD].Payload[1]);
  
      // Get current message state 
     _cmdMessageState := GetHalfeByteLo(Value := Register[_regIdx].Response[ACTIVE_CMD].Payload[0]);

  
      // Create log entry
      CreateLogMessagePara3( Timestamp   := SystemTime,
                             MessageType := MessageType.CMD,
                             Severity    := Severity.INFO,
                             MessageCode := 0,
                             MessageText := 'ACR-ID [{1}]: Deleted ACR-Entry of CmdType <{2}> with State = {3}, because of Final-State was reached',
                             Para1       :=  DINT_TO_STRING(_regIdx),
                             Para2       :=  CMD_TYPE_TO_STRING(_cmdType),
                             Para3       :=  CMD_MESSAGE_STATE_TO_STRING(_cmdMessageState));
  
                             
      // delete register entry                              
      Register[_regIdx] := EMPTY_ACR_ENTRY;

      // decrement current used register counter
      CurrentAcrUsageCount := CurrentAcrUsageCount - 1;                           
    END_IF
  END_IF
END_FOR


